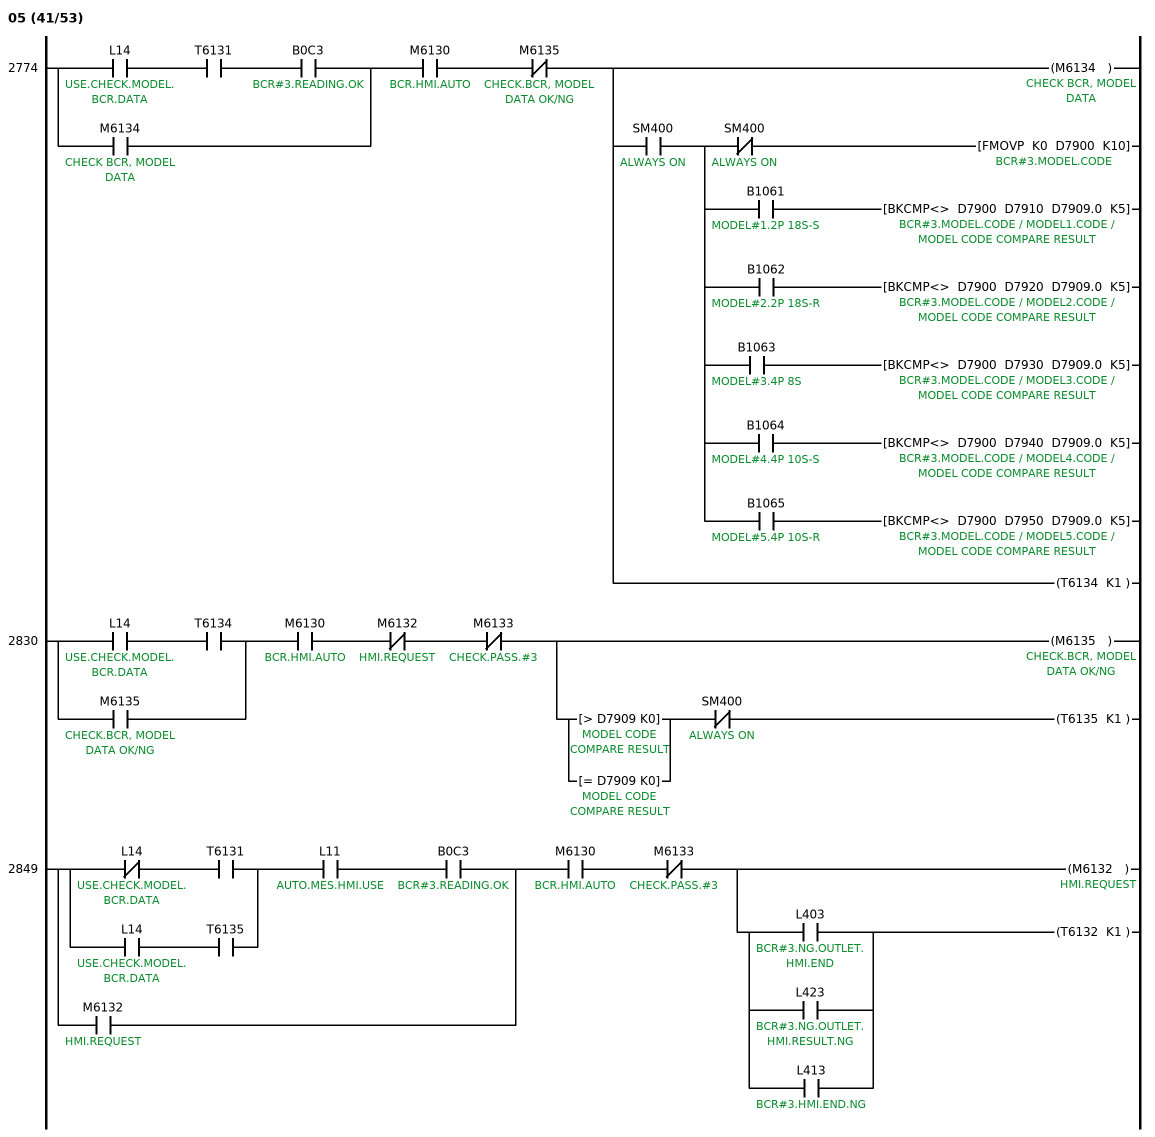
2774  LD      L14  ; USE.CHECK.MODEL.BCR.DATA
      AND     T6131
      AND     B0C3  ; BCR#3.READING.OK
      OR      M6134  ; CHECK BCR, MODEL DATA
      AND     M6130  ; BCR.HMI.AUTO
      ANI     M6135  ; CHECK.BCR, MODEL DATA OK/NG
      OUT     M6134  ; CHECK BCR, MODEL DATA
      MPS
      AND     SM400  ; ALWAYS ON
      MPS
      ANI     SM400  ; ALWAYS ON
      FMOVP   K0 D7900 K10  ; BCR#3.MODEL.CODE
      MRD
      AND     B1061  ; MODEL#1.2P 18S-S
      BKCMP<> D7900 D7910 D7909.0 K5  ; MODEL1.CODE / MODEL CODE COMPARE RESULT
      MRD
      AND     B1062  ; MODEL#2.2P 18S-R
      BKCMP<> D7900 D7920 D7909.0 K5  ; MODEL2.CODE
      MRD
      AND     B1063  ; MODEL#3.4P 8S
      BKCMP<> D7900 D7930 D7909.0 K5  ; MODEL3.CODE
      MRD
      AND     B1064  ; MODEL#4.4P 10S-S
      BKCMP<> D7900 D7940 D7909.0 K5  ; MODEL4.CODE
      MPP
      AND     B1065  ; MODEL#5.4P 10S-R
      BKCMP<> D7900 D7950 D7909.0 K5  ; MODEL5.CODE
      MPP
      OUT     T6134 K1
2830  LD      L14  ; USE.CHECK.MODEL.BCR.DATA
      AND     T6134
      OR      M6135  ; CHECK.BCR, MODEL DATA OK/NG
      AND     M6130  ; BCR.HMI.AUTO
      ANI     M6132  ; HMI.REQUEST
      ANI     M6133  ; CHECK.PASS.#3
      OUT     M6135  ; CHECK.BCR, MODEL DATA OK/NG
      LD>     D7909 K0  ; MODEL CODE COMPARE RESULT
      OR=     D7909 K0  ; MODEL CODE COMPARE RESULT
      ANB
      ANI     SM400  ; ALWAYS ON
      OUT     T6135 K1
2849  LDI     L14  ; USE.CHECK.MODEL.BCR.DATA
      AND     T6131
      LD      L14  ; USE.CHECK.MODEL.BCR.DATA
      AND     T6135
      ORB
      AND     L11  ; AUTO.MES.HMI.USE
      AND     B0C3  ; BCR#3.READING.OK
      OR      M6132  ; HMI.REQUEST
      AND     M6130  ; BCR.HMI.AUTO
      ANI     M6133  ; CHECK.PASS.#3
      OUT     M6132  ; HMI.REQUEST
      LD      L403  ; BCR#3.NG.OUTLET.HMI.END
      OR      L423  ; BCR#3.NG.OUTLET.HMI.RESULT.NG
      OR      L413  ; BCR#3.HMI.END.NG
      ANB
      OUT     T6132 K1
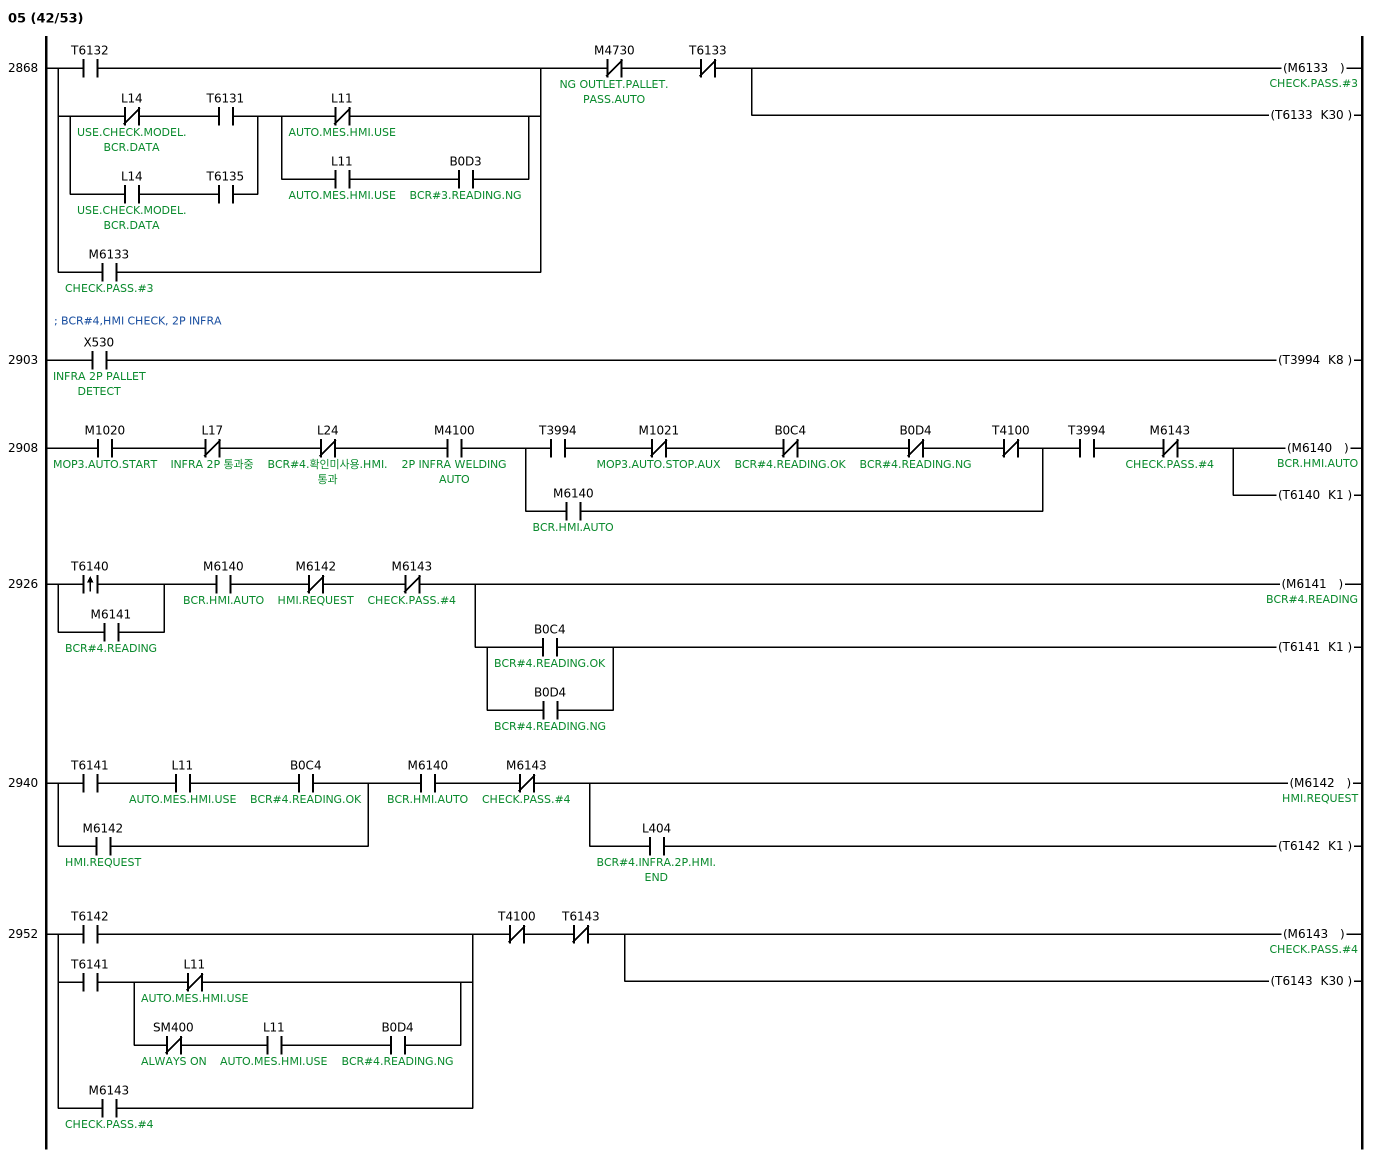
2868  LD      T6132
      LDI     L14  ; USE.CHECK.MODEL.BCR.DATA
      AND     T6131
      LD      L14  ; USE.CHECK.MODEL.BCR.DATA
      AND     T6135
      ORB
      LDI     L11  ; AUTO.MES.HMI.USE
      LD      L11  ; AUTO.MES.HMI.USE
      AND     B0D3  ; BCR#3.READING.NG
      ORB
      ANB
      ORB
      OR      M6133  ; CHECK.PASS.#3
      ANI     M4730  ; NG OUTLET.PALLET.PASS.AUTO
      ANI     T6133
      OUT     M6133  ; CHECK.PASS.#3
      OUT     T6133 K30
; BCR#4,HMI CHECK, 2P INFRA
2903  LD      X530  ; INFRA 2P PALLET DETECT
      OUT     T3994 K8
2908  LD      M1020  ; MOP3.AUTO.START
      ANI     L17  ; INFRA 2P 통과중
      ANI     L24  ; BCR#4.확인미사용.HMI.통과
      AND     M4100  ; 2P INFRA WELDING AUTO
      LD      T3994
      ANI     M1021  ; MOP3.AUTO.STOP.AUX
      ANI     B0C4  ; BCR#4.READING.OK
      ANI     B0D4  ; BCR#4.READING.NG
      ANI     T4100
      OR      M6140  ; BCR.HMI.AUTO
      ANB
      AND     T3994
      ANI     M6143  ; CHECK.PASS.#4
      OUT     M6140  ; BCR.HMI.AUTO
      OUT     T6140 K1
2926  LDP     T6140
      OR      M6141  ; BCR#4.READING
      AND     M6140  ; BCR.HMI.AUTO
      ANI     M6142  ; HMI.REQUEST
      ANI     M6143  ; CHECK.PASS.#4
      OUT     M6141  ; BCR#4.READING
      LD      B0C4  ; BCR#4.READING.OK
      OR      B0D4  ; BCR#4.READING.NG
      ANB
      OUT     T6141 K1
2940  LD      T6141
      AND     L11  ; AUTO.MES.HMI.USE
      AND     B0C4  ; BCR#4.READING.OK
      OR      M6142  ; HMI.REQUEST
      AND     M6140  ; BCR.HMI.AUTO
      ANI     M6143  ; CHECK.PASS.#4
      OUT     M6142  ; HMI.REQUEST
      AND     L404  ; BCR#4.INFRA.2P.HMI.END
      OUT     T6142 K1
2952  LD      T6142
      LD      T6141
      LDI     L11  ; AUTO.MES.HMI.USE
      LDI     SM400  ; ALWAYS ON
      AND     L11  ; AUTO.MES.HMI.USE
      AND     B0D4  ; BCR#4.READING.NG
      ORB
      ANB
      ORB
      OR      M6143  ; CHECK.PASS.#4
      ANI     T4100
      ANI     T6143
      OUT     M6143  ; CHECK.PASS.#4
      OUT     T6143 K30
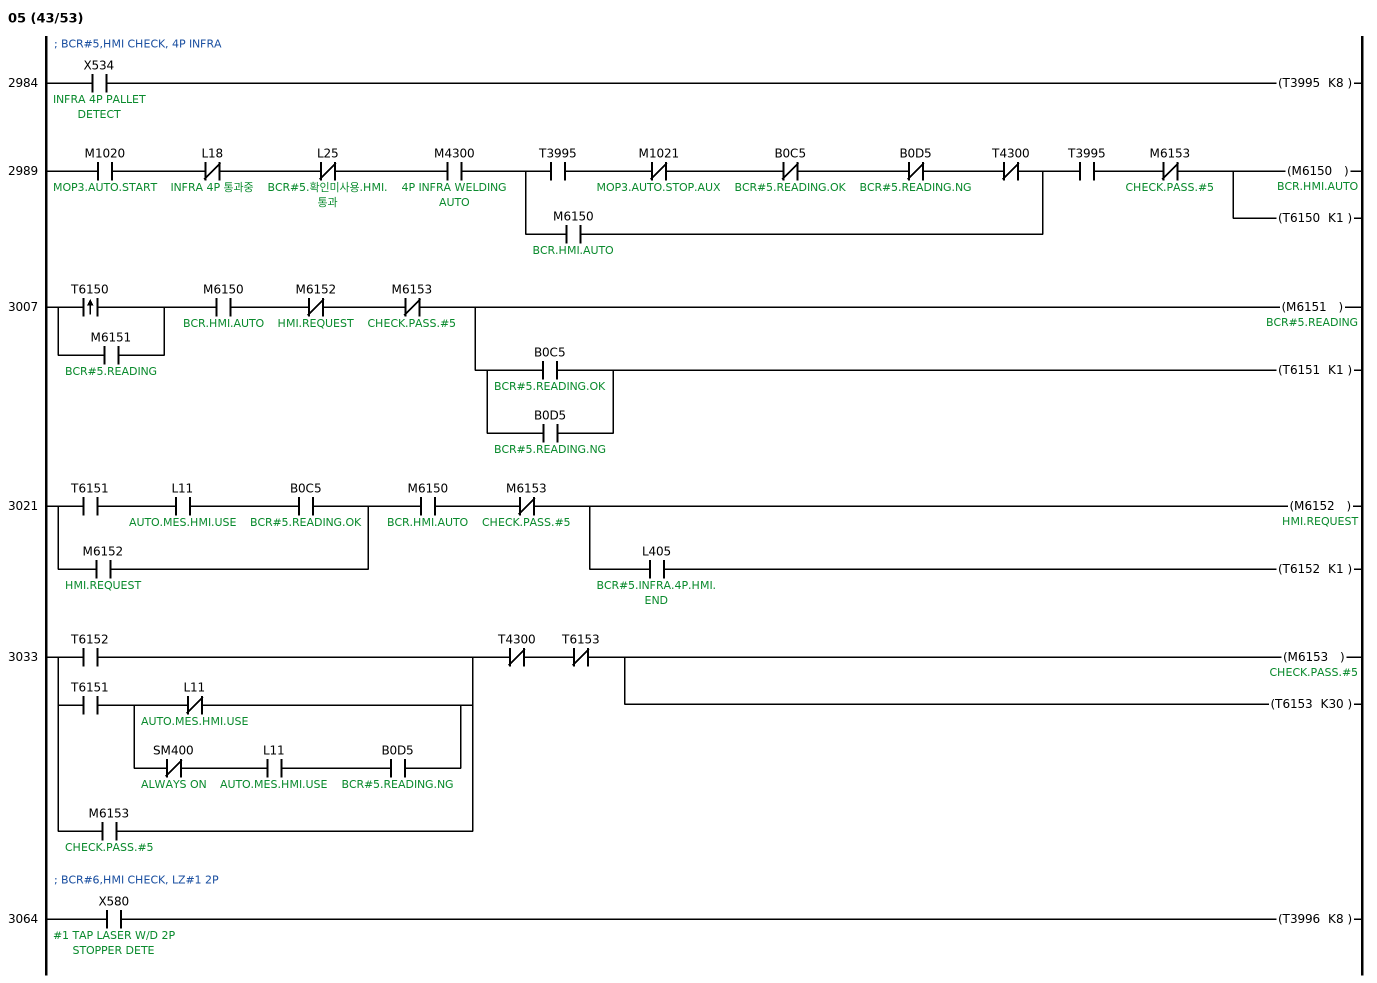
; BCR#5,HMI CHECK, 4P INFRA
2984  LD      X534  ; INFRA 4P PALLET DETECT
      OUT     T3995 K8
2989  LD      M1020  ; MOP3.AUTO.START
      ANI     L18  ; INFRA 4P 통과중
      ANI     L25  ; BCR#5.확인미사용.HMI.통과
      AND     M4300  ; 4P INFRA WELDING AUTO
      LD      T3995
      ANI     M1021  ; MOP3.AUTO.STOP.AUX
      ANI     B0C5  ; BCR#5.READING.OK
      ANI     B0D5  ; BCR#5.READING.NG
      ANI     T4300
      OR      M6150  ; BCR.HMI.AUTO
      ANB
      AND     T3995
      ANI     M6153  ; CHECK.PASS.#5
      OUT     M6150  ; BCR.HMI.AUTO
      OUT     T6150 K1
3007  LDP     T6150
      OR      M6151  ; BCR#5.READING
      AND     M6150  ; BCR.HMI.AUTO
      ANI     M6152  ; HMI.REQUEST
      ANI     M6153  ; CHECK.PASS.#5
      OUT     M6151  ; BCR#5.READING
      LD      B0C5  ; BCR#5.READING.OK
      OR      B0D5  ; BCR#5.READING.NG
      ANB
      OUT     T6151 K1
3021  LD      T6151
      AND     L11  ; AUTO.MES.HMI.USE
      AND     B0C5  ; BCR#5.READING.OK
      OR      M6152  ; HMI.REQUEST
      AND     M6150  ; BCR.HMI.AUTO
      ANI     M6153  ; CHECK.PASS.#5
      OUT     M6152  ; HMI.REQUEST
      AND     L405  ; BCR#5.INFRA.4P.HMI.END
      OUT     T6152 K1
3033  LD      T6152
      LD      T6151
      LDI     L11  ; AUTO.MES.HMI.USE
      LDI     SM400  ; ALWAYS ON
      AND     L11  ; AUTO.MES.HMI.USE
      AND     B0D5  ; BCR#5.READING.NG
      ORB
      ANB
      ORB
      OR      M6153  ; CHECK.PASS.#5
      ANI     T4300
      ANI     T6153
      OUT     M6153  ; CHECK.PASS.#5
      OUT     T6153 K30
; BCR#6,HMI CHECK, LZ#1 2P
3064  LD      X580  ; #1 TAP LASER W/D 2P STOPPER DETE
      OUT     T3996 K8
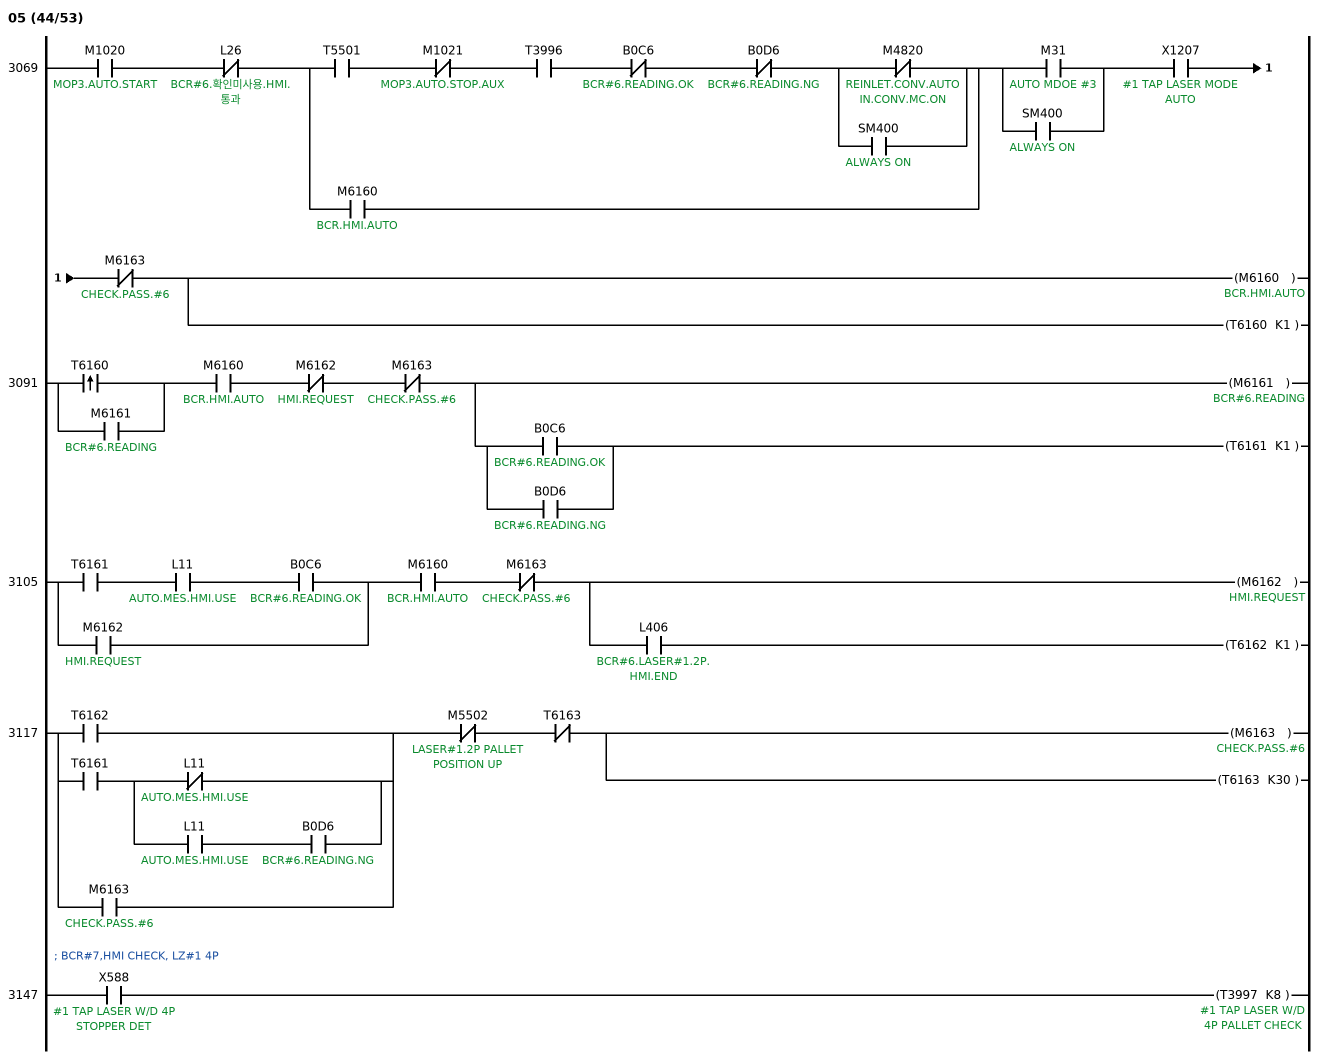
3069  LD      M1020  ; MOP3.AUTO.START
      ANI     L26  ; BCR#6.확인미사용.HMI.통과
      LD      T5501
      ANI     M1021  ; MOP3.AUTO.STOP.AUX
      AND     T3996
      ANI     B0C6  ; BCR#6.READING.OK
      ANI     B0D6  ; BCR#6.READING.NG
      LDI     M4820  ; REINLET.CONV.AUTO IN.CONV.MC.ON
      OR      SM400  ; ALWAYS ON
      ANB
      OR      M6160  ; BCR.HMI.AUTO
      ANB
      LD      M31  ; AUTO MDOE #3
      OR      SM400  ; ALWAYS ON
      ANB
      AND     X1207  ; #1 TAP LASER MODE AUTO
      ANI     M6163  ; CHECK.PASS.#6
      OUT     M6160  ; BCR.HMI.AUTO
      OUT     T6160 K1
3091  LDP     T6160
      OR      M6161  ; BCR#6.READING
      AND     M6160  ; BCR.HMI.AUTO
      ANI     M6162  ; HMI.REQUEST
      ANI     M6163  ; CHECK.PASS.#6
      OUT     M6161  ; BCR#6.READING
      LD      B0C6  ; BCR#6.READING.OK
      OR      B0D6  ; BCR#6.READING.NG
      ANB
      OUT     T6161 K1
3105  LD      T6161
      AND     L11  ; AUTO.MES.HMI.USE
      AND     B0C6  ; BCR#6.READING.OK
      OR      M6162  ; HMI.REQUEST
      AND     M6160  ; BCR.HMI.AUTO
      ANI     M6163  ; CHECK.PASS.#6
      OUT     M6162  ; HMI.REQUEST
      AND     L406  ; BCR#6.LASER#1.2P.HMI.END
      OUT     T6162 K1
3117  LD      T6162
      LD      T6161
      LDI     L11  ; AUTO.MES.HMI.USE
      LD      L11  ; AUTO.MES.HMI.USE
      AND     B0D6  ; BCR#6.READING.NG
      ORB
      ANB
      ORB
      OR      M6163  ; CHECK.PASS.#6
      ANI     M5502  ; LASER#1.2P PALLET POSITION UP
      ANI     T6163
      OUT     M6163  ; CHECK.PASS.#6
      OUT     T6163 K30
; BCR#7,HMI CHECK, LZ#1 4P
3147  LD      X588  ; #1 TAP LASER W/D 4P STOPPER DET
      OUT     T3997 K8  ; #1 TAP LASER W/D 4P PALLET CHECK
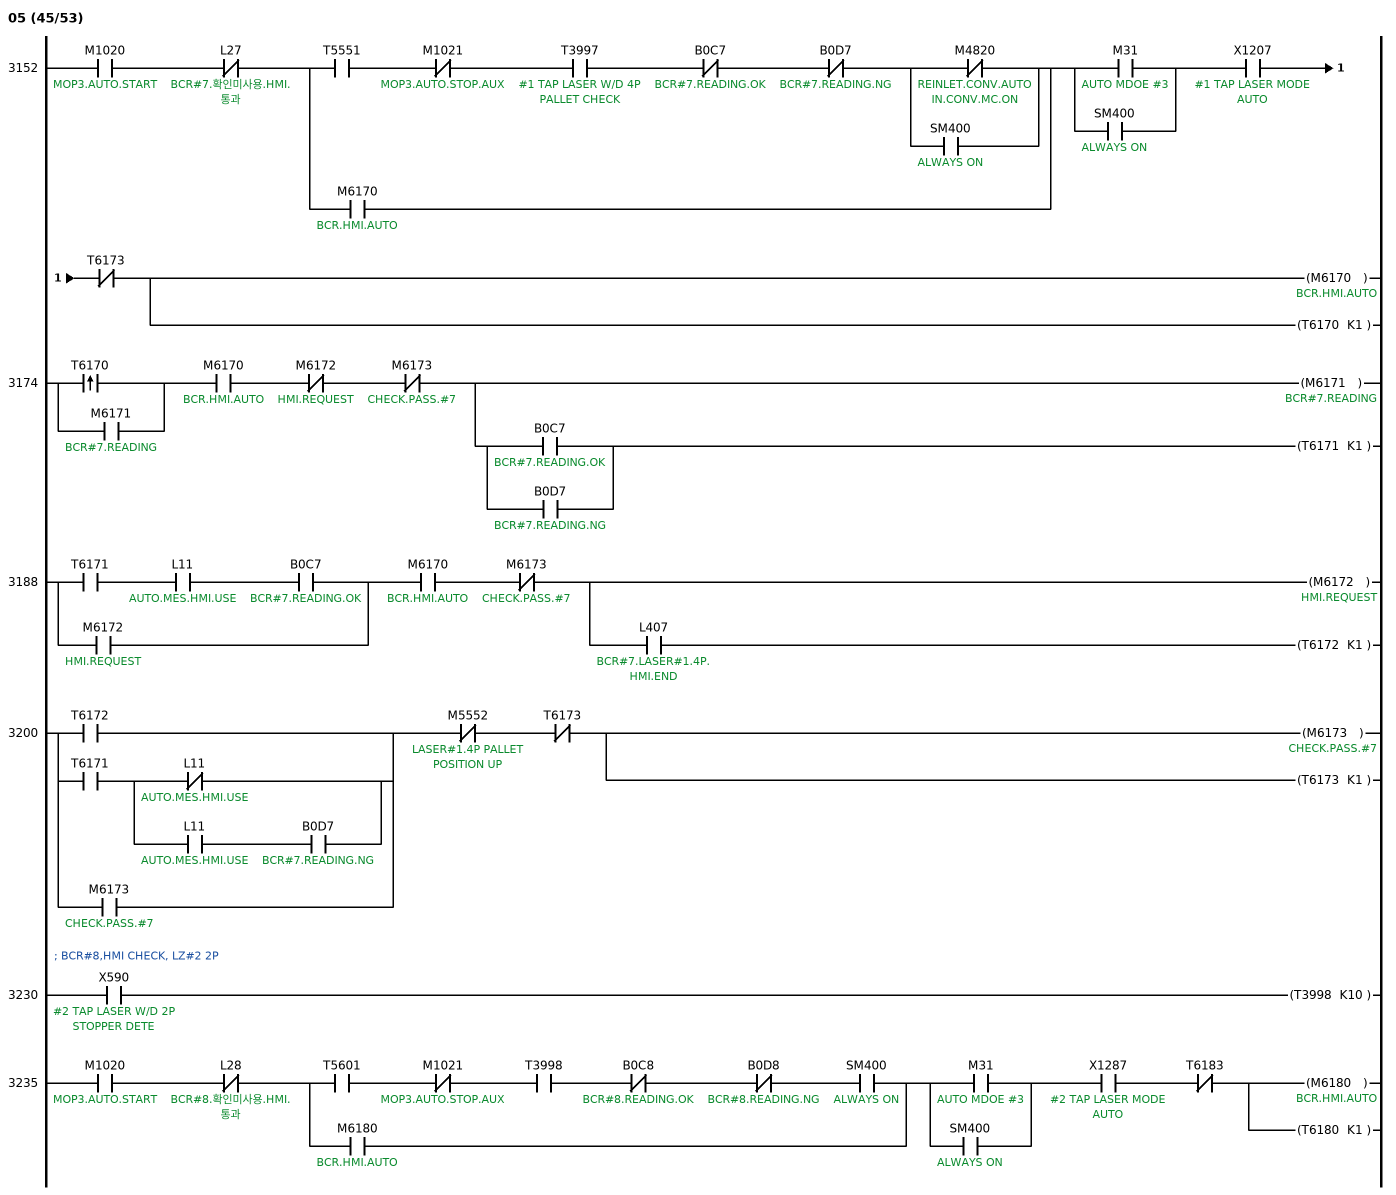
3152  LD      M1020  ; MOP3.AUTO.START
      ANI     L27  ; BCR#7.확인미사용.HMI.통과
      LD      T5551
      ANI     M1021  ; MOP3.AUTO.STOP.AUX
      AND     T3997  ; #1 TAP LASER W/D 4P PALLET CHECK
      ANI     B0C7  ; BCR#7.READING.OK
      ANI     B0D7  ; BCR#7.READING.NG
      LDI     M4820  ; REINLET.CONV.AUTO IN.CONV.MC.ON
      OR      SM400  ; ALWAYS ON
      ANB
      OR      M6170  ; BCR.HMI.AUTO
      ANB
      LD      M31  ; AUTO MDOE #3
      OR      SM400  ; ALWAYS ON
      ANB
      AND     X1207  ; #1 TAP LASER MODE AUTO
      ANI     T6173
      OUT     M6170  ; BCR.HMI.AUTO
      OUT     T6170 K1
3174  LDP     T6170
      OR      M6171  ; BCR#7.READING
      AND     M6170  ; BCR.HMI.AUTO
      ANI     M6172  ; HMI.REQUEST
      ANI     M6173  ; CHECK.PASS.#7
      OUT     M6171  ; BCR#7.READING
      LD      B0C7  ; BCR#7.READING.OK
      OR      B0D7  ; BCR#7.READING.NG
      ANB
      OUT     T6171 K1
3188  LD      T6171
      AND     L11  ; AUTO.MES.HMI.USE
      AND     B0C7  ; BCR#7.READING.OK
      OR      M6172  ; HMI.REQUEST
      AND     M6170  ; BCR.HMI.AUTO
      ANI     M6173  ; CHECK.PASS.#7
      OUT     M6172  ; HMI.REQUEST
      AND     L407  ; BCR#7.LASER#1.4P.HMI.END
      OUT     T6172 K1
3200  LD      T6172
      LD      T6171
      LDI     L11  ; AUTO.MES.HMI.USE
      LD      L11  ; AUTO.MES.HMI.USE
      AND     B0D7  ; BCR#7.READING.NG
      ORB
      ANB
      ORB
      OR      M6173  ; CHECK.PASS.#7
      ANI     M5552  ; LASER#1.4P PALLET POSITION UP
      ANI     T6173
      OUT     M6173  ; CHECK.PASS.#7
      OUT     T6173 K1
; BCR#8,HMI CHECK, LZ#2 2P
3230  LD      X590  ; #2 TAP LASER W/D 2P STOPPER DETE
      OUT     T3998 K10
3235  LD      M1020  ; MOP3.AUTO.START
      ANI     L28  ; BCR#8.확인미사용.HMI.통과
      LD      T5601
      ANI     M1021  ; MOP3.AUTO.STOP.AUX
      AND     T3998
      ANI     B0C8  ; BCR#8.READING.OK
      ANI     B0D8  ; BCR#8.READING.NG
      AND     SM400  ; ALWAYS ON
      OR      M6180  ; BCR.HMI.AUTO
      ANB
      LD      M31  ; AUTO MDOE #3
      OR      SM400  ; ALWAYS ON
      ANB
      AND     X1287  ; #2 TAP LASER MODE AUTO
      ANI     T6183
      OUT     M6180  ; BCR.HMI.AUTO
      OUT     T6180 K1
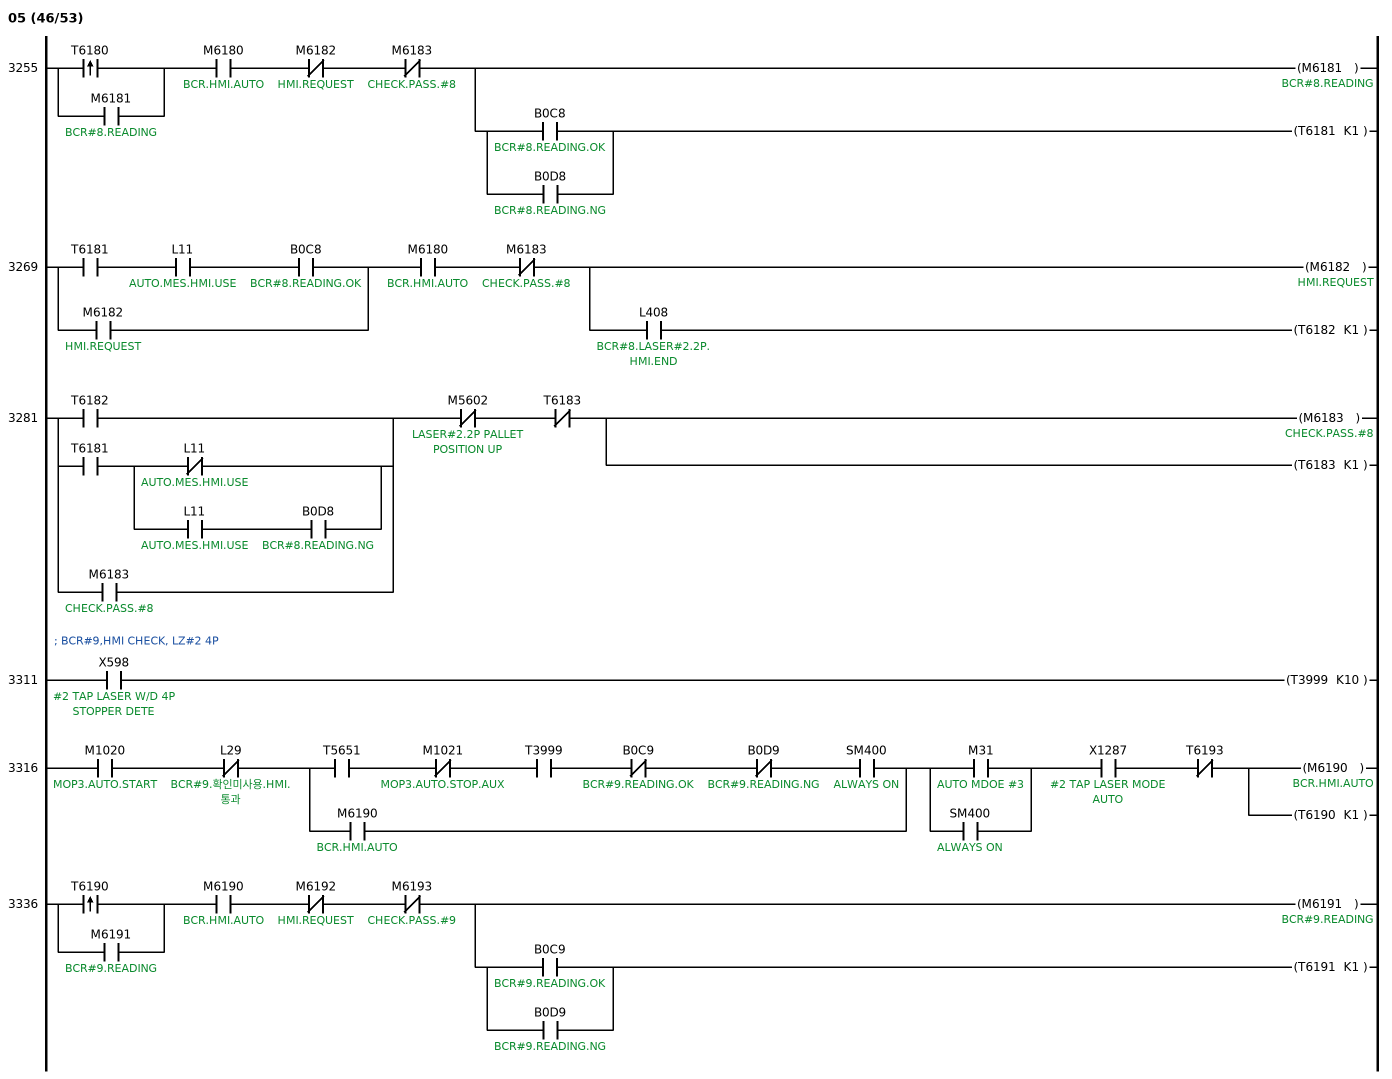
3255  LDP     T6180
      OR      M6181  ; BCR#8.READING
      AND     M6180  ; BCR.HMI.AUTO
      ANI     M6182  ; HMI.REQUEST
      ANI     M6183  ; CHECK.PASS.#8
      OUT     M6181  ; BCR#8.READING
      LD      B0C8  ; BCR#8.READING.OK
      OR      B0D8  ; BCR#8.READING.NG
      ANB
      OUT     T6181 K1
3269  LD      T6181
      AND     L11  ; AUTO.MES.HMI.USE
      AND     B0C8  ; BCR#8.READING.OK
      OR      M6182  ; HMI.REQUEST
      AND     M6180  ; BCR.HMI.AUTO
      ANI     M6183  ; CHECK.PASS.#8
      OUT     M6182  ; HMI.REQUEST
      AND     L408  ; BCR#8.LASER#2.2P.HMI.END
      OUT     T6182 K1
3281  LD      T6182
      LD      T6181
      LDI     L11  ; AUTO.MES.HMI.USE
      LD      L11  ; AUTO.MES.HMI.USE
      AND     B0D8  ; BCR#8.READING.NG
      ORB
      ANB
      ORB
      OR      M6183  ; CHECK.PASS.#8
      ANI     M5602  ; LASER#2.2P PALLET POSITION UP
      ANI     T6183
      OUT     M6183  ; CHECK.PASS.#8
      OUT     T6183 K1
; BCR#9,HMI CHECK, LZ#2 4P
3311  LD      X598  ; #2 TAP LASER W/D 4P STOPPER DETE
      OUT     T3999 K10
3316  LD      M1020  ; MOP3.AUTO.START
      ANI     L29  ; BCR#9.확인미사용.HMI.통과
      LD      T5651
      ANI     M1021  ; MOP3.AUTO.STOP.AUX
      AND     T3999
      ANI     B0C9  ; BCR#9.READING.OK
      ANI     B0D9  ; BCR#9.READING.NG
      AND     SM400  ; ALWAYS ON
      OR      M6190  ; BCR.HMI.AUTO
      ANB
      LD      M31  ; AUTO MDOE #3
      OR      SM400  ; ALWAYS ON
      ANB
      AND     X1287  ; #2 TAP LASER MODE AUTO
      ANI     T6193
      OUT     M6190  ; BCR.HMI.AUTO
      OUT     T6190 K1
3336  LDP     T6190
      OR      M6191  ; BCR#9.READING
      AND     M6190  ; BCR.HMI.AUTO
      ANI     M6192  ; HMI.REQUEST
      ANI     M6193  ; CHECK.PASS.#9
      OUT     M6191  ; BCR#9.READING
      LD      B0C9  ; BCR#9.READING.OK
      OR      B0D9  ; BCR#9.READING.NG
      ANB
      OUT     T6191 K1
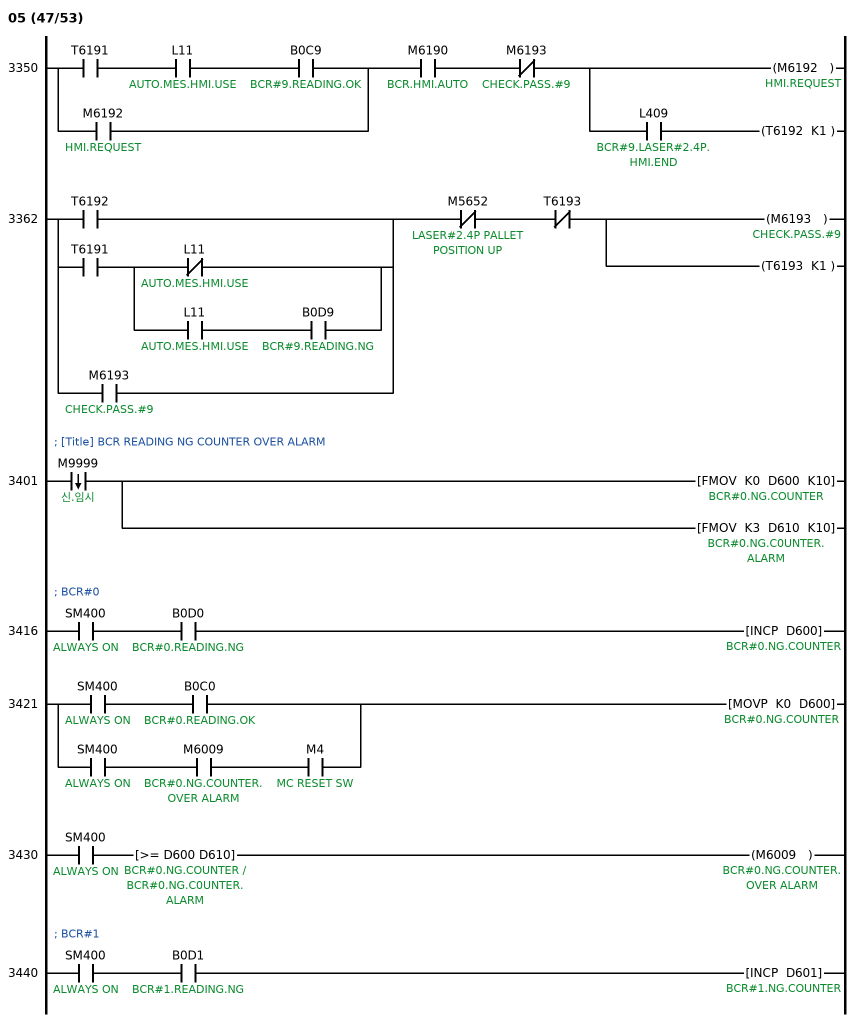
3350  LD      T6191
      AND     L11  ; AUTO.MES.HMI.USE
      AND     B0C9  ; BCR#9.READING.OK
      OR      M6192  ; HMI.REQUEST
      AND     M6190  ; BCR.HMI.AUTO
      ANI     M6193  ; CHECK.PASS.#9
      OUT     M6192  ; HMI.REQUEST
      AND     L409  ; BCR#9.LASER#2.4P.HMI.END
      OUT     T6192 K1
3362  LD      T6192
      LD      T6191
      LDI     L11  ; AUTO.MES.HMI.USE
      LD      L11  ; AUTO.MES.HMI.USE
      AND     B0D9  ; BCR#9.READING.NG
      ORB
      ANB
      ORB
      OR      M6193  ; CHECK.PASS.#9
      ANI     M5652  ; LASER#2.4P PALLET POSITION UP
      ANI     T6193
      OUT     M6193  ; CHECK.PASS.#9
      OUT     T6193 K1
; [Title] BCR READING NG COUNTER OVER ALARM
3401  LDF     M9999  ; 신.임시
      FMOV    K0 D600 K10  ; BCR#0.NG.COUNTER
      FMOV    K3 D610 K10  ; BCR#0.NG.C0UNTER.ALARM
; BCR#0
3416  LD      SM400  ; ALWAYS ON
      AND     B0D0  ; BCR#0.READING.NG
      INCP    D600
3421  LD      SM400  ; ALWAYS ON
      AND     B0C0  ; BCR#0.READING.OK
      LD      SM400  ; ALWAYS ON
      AND     M6009  ; BCR#0.NG.COUNTER.OVER ALARM
      AND     M4  ; MC RESET SW
      ORB
      MOVP    K0 D600
3430  LD      SM400  ; ALWAYS ON
      AND>=   D600 D610  ; BCR#0.NG.COUNTER / BCR#0.NG.C0UNTER.ALARM
      OUT     M6009  ; BCR#0.NG.COUNTER.OVER ALARM
; BCR#1
3440  LD      SM400  ; ALWAYS ON
      AND     B0D1  ; BCR#1.READING.NG
      INCP    D601  ; BCR#1.NG.COUNTER
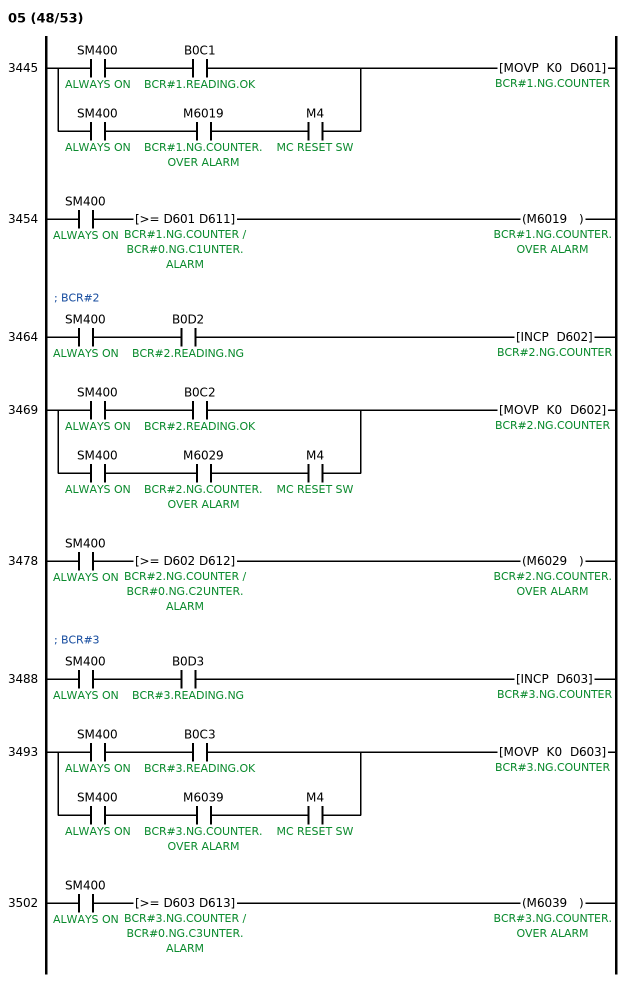
3445  LD      SM400  ; ALWAYS ON
      AND     B0C1  ; BCR#1.READING.OK
      LD      SM400  ; ALWAYS ON
      AND     M6019  ; BCR#1.NG.COUNTER.OVER ALARM
      AND     M4  ; MC RESET SW
      ORB
      MOVP    K0 D601
3454  LD      SM400  ; ALWAYS ON
      AND>=   D601 D611  ; BCR#1.NG.COUNTER / BCR#0.NG.C1UNTER.ALARM
      OUT     M6019  ; BCR#1.NG.COUNTER.OVER ALARM
; BCR#2
3464  LD      SM400  ; ALWAYS ON
      AND     B0D2  ; BCR#2.READING.NG
      INCP    D602  ; BCR#2.NG.COUNTER
3469  LD      SM400  ; ALWAYS ON
      AND     B0C2  ; BCR#2.READING.OK
      LD      SM400  ; ALWAYS ON
      AND     M6029  ; BCR#2.NG.COUNTER.OVER ALARM
      AND     M4  ; MC RESET SW
      ORB
      MOVP    K0 D602
3478  LD      SM400  ; ALWAYS ON
      AND>=   D602 D612  ; BCR#2.NG.COUNTER / BCR#0.NG.C2UNTER.ALARM
      OUT     M6029  ; BCR#2.NG.COUNTER.OVER ALARM
; BCR#3
3488  LD      SM400  ; ALWAYS ON
      AND     B0D3  ; BCR#3.READING.NG
      INCP    D603  ; BCR#3.NG.COUNTER
3493  LD      SM400  ; ALWAYS ON
      AND     B0C3  ; BCR#3.READING.OK
      LD      SM400  ; ALWAYS ON
      AND     M6039  ; BCR#3.NG.COUNTER.OVER ALARM
      AND     M4  ; MC RESET SW
      ORB
      MOVP    K0 D603
3502  LD      SM400  ; ALWAYS ON
      AND>=   D603 D613  ; BCR#3.NG.COUNTER / BCR#0.NG.C3UNTER.ALARM
      OUT     M6039  ; BCR#3.NG.COUNTER.OVER ALARM
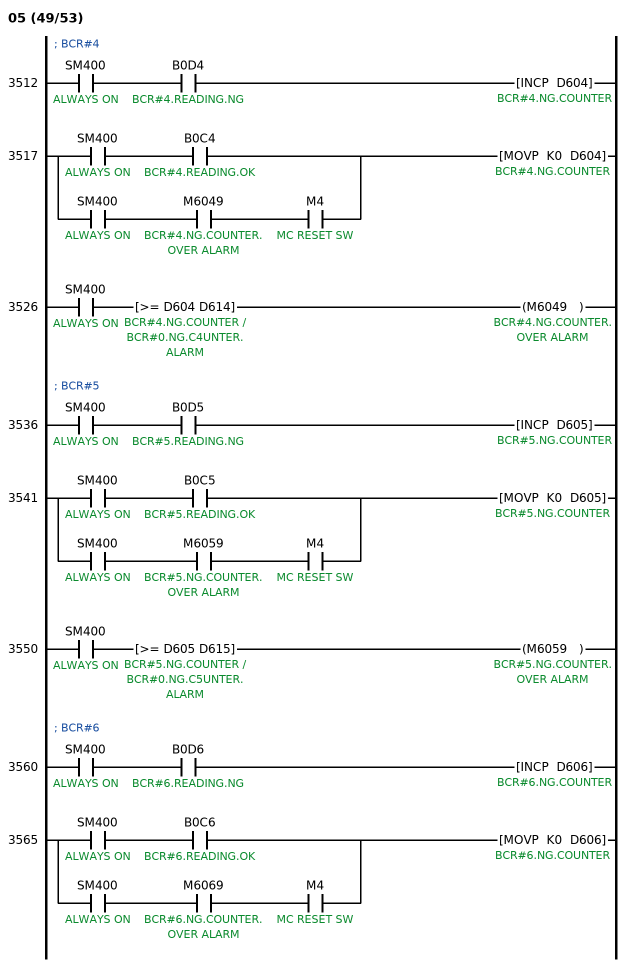
; BCR#4
3512  LD      SM400  ; ALWAYS ON
      AND     B0D4  ; BCR#4.READING.NG
      INCP    D604  ; BCR#4.NG.COUNTER
3517  LD      SM400  ; ALWAYS ON
      AND     B0C4  ; BCR#4.READING.OK
      LD      SM400  ; ALWAYS ON
      AND     M6049  ; BCR#4.NG.COUNTER.OVER ALARM
      AND     M4  ; MC RESET SW
      ORB
      MOVP    K0 D604
3526  LD      SM400  ; ALWAYS ON
      AND>=   D604 D614  ; BCR#4.NG.COUNTER / BCR#0.NG.C4UNTER.ALARM
      OUT     M6049  ; BCR#4.NG.COUNTER.OVER ALARM
; BCR#5
3536  LD      SM400  ; ALWAYS ON
      AND     B0D5  ; BCR#5.READING.NG
      INCP    D605  ; BCR#5.NG.COUNTER
3541  LD      SM400  ; ALWAYS ON
      AND     B0C5  ; BCR#5.READING.OK
      LD      SM400  ; ALWAYS ON
      AND     M6059  ; BCR#5.NG.COUNTER.OVER ALARM
      AND     M4  ; MC RESET SW
      ORB
      MOVP    K0 D605
3550  LD      SM400  ; ALWAYS ON
      AND>=   D605 D615  ; BCR#5.NG.COUNTER / BCR#0.NG.C5UNTER.ALARM
      OUT     M6059  ; BCR#5.NG.COUNTER.OVER ALARM
; BCR#6
3560  LD      SM400  ; ALWAYS ON
      AND     B0D6  ; BCR#6.READING.NG
      INCP    D606  ; BCR#6.NG.COUNTER
3565  LD      SM400  ; ALWAYS ON
      AND     B0C6  ; BCR#6.READING.OK
      LD      SM400  ; ALWAYS ON
      AND     M6069  ; BCR#6.NG.COUNTER.OVER ALARM
      AND     M4  ; MC RESET SW
      ORB
      MOVP    K0 D606
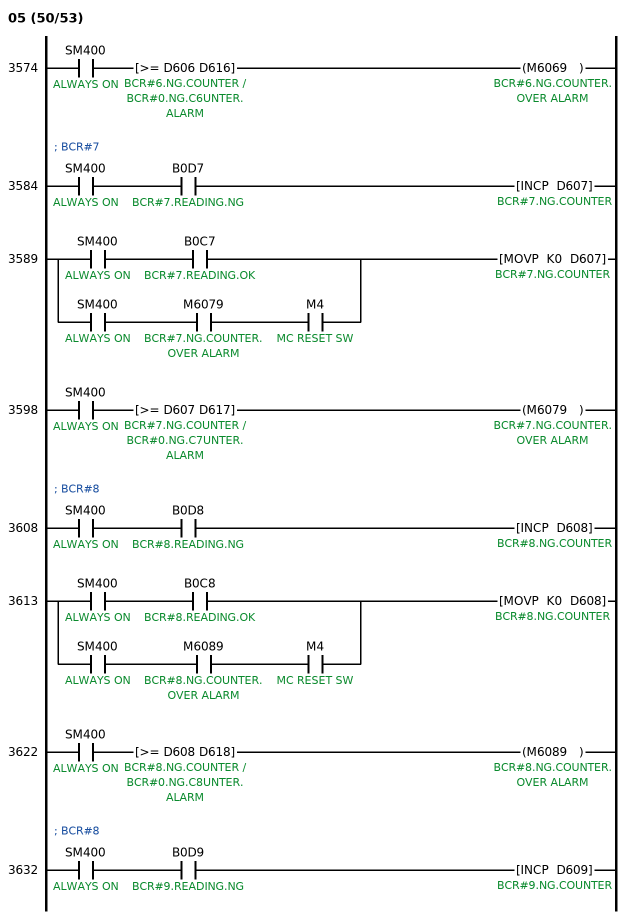
3574  LD      SM400  ; ALWAYS ON
      AND>=   D606 D616  ; BCR#6.NG.COUNTER / BCR#0.NG.C6UNTER.ALARM
      OUT     M6069  ; BCR#6.NG.COUNTER.OVER ALARM
; BCR#7
3584  LD      SM400  ; ALWAYS ON
      AND     B0D7  ; BCR#7.READING.NG
      INCP    D607  ; BCR#7.NG.COUNTER
3589  LD      SM400  ; ALWAYS ON
      AND     B0C7  ; BCR#7.READING.OK
      LD      SM400  ; ALWAYS ON
      AND     M6079  ; BCR#7.NG.COUNTER.OVER ALARM
      AND     M4  ; MC RESET SW
      ORB
      MOVP    K0 D607
3598  LD      SM400  ; ALWAYS ON
      AND>=   D607 D617  ; BCR#7.NG.COUNTER / BCR#0.NG.C7UNTER.ALARM
      OUT     M6079  ; BCR#7.NG.COUNTER.OVER ALARM
; BCR#8
3608  LD      SM400  ; ALWAYS ON
      AND     B0D8  ; BCR#8.READING.NG
      INCP    D608  ; BCR#8.NG.COUNTER
3613  LD      SM400  ; ALWAYS ON
      AND     B0C8  ; BCR#8.READING.OK
      LD      SM400  ; ALWAYS ON
      AND     M6089  ; BCR#8.NG.COUNTER.OVER ALARM
      AND     M4  ; MC RESET SW
      ORB
      MOVP    K0 D608
3622  LD      SM400  ; ALWAYS ON
      AND>=   D608 D618  ; BCR#8.NG.COUNTER / BCR#0.NG.C8UNTER.ALARM
      OUT     M6089  ; BCR#8.NG.COUNTER.OVER ALARM
; BCR#8
3632  LD      SM400  ; ALWAYS ON
      AND     B0D9  ; BCR#9.READING.NG
      INCP    D609  ; BCR#9.NG.COUNTER
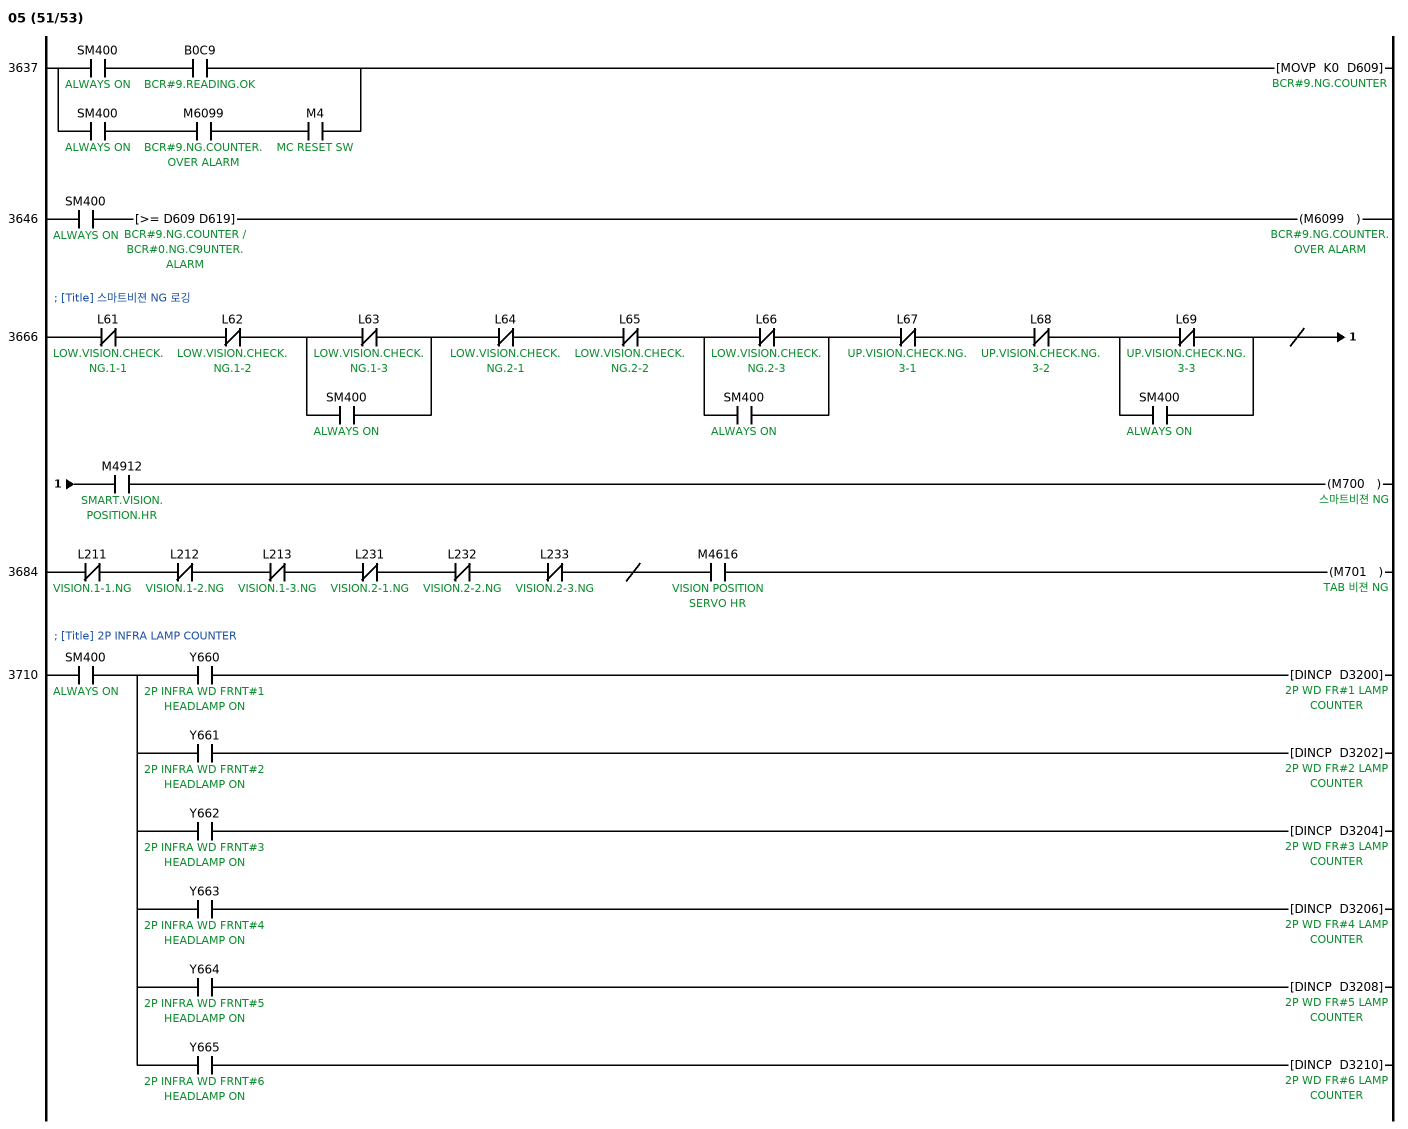
3637  LD      SM400  ; ALWAYS ON
      AND     B0C9  ; BCR#9.READING.OK
      LD      SM400  ; ALWAYS ON
      AND     M6099  ; BCR#9.NG.COUNTER.OVER ALARM
      AND     M4  ; MC RESET SW
      ORB
      MOVP    K0 D609
3646  LD      SM400  ; ALWAYS ON
      AND>=   D609 D619  ; BCR#9.NG.COUNTER / BCR#0.NG.C9UNTER.ALARM
      OUT     M6099  ; BCR#9.NG.COUNTER.OVER ALARM
; [Title] 스마트비젼 NG 로깅
3666  LDI     L61  ; LOW.VISION.CHECK.NG.1-1
      ANI     L62  ; LOW.VISION.CHECK.NG.1-2
      LDI     L63  ; LOW.VISION.CHECK.NG.1-3
      OR      SM400  ; ALWAYS ON
      ANB
      ANI     L64  ; LOW.VISION.CHECK.NG.2-1
      ANI     L65  ; LOW.VISION.CHECK.NG.2-2
      LDI     L66  ; LOW.VISION.CHECK.NG.2-3
      OR      SM400  ; ALWAYS ON
      ANB
      ANI     L67  ; UP.VISION.CHECK.NG.3-1
      ANI     L68  ; UP.VISION.CHECK.NG.3-2
      LDI     L69  ; UP.VISION.CHECK.NG.3-3
      OR      SM400  ; ALWAYS ON
      ANB
      INV
      AND     M4912  ; SMART.VISION.POSITION.HR
      OUT     M700  ; 스마트비젼 NG
3684  LDI     L211  ; VISION.1-1.NG
      ANI     L212  ; VISION.1-2.NG
      ANI     L213  ; VISION.1-3.NG
      ANI     L231  ; VISION.2-1.NG
      ANI     L232  ; VISION.2-2.NG
      ANI     L233  ; VISION.2-3.NG
      INV
      AND     M4616  ; VISION POSITION SERVO HR
      OUT     M701  ; TAB 비젼 NG
; [Title] 2P INFRA LAMP COUNTER
3710  LD      SM400  ; ALWAYS ON
      MPS
      AND     Y660  ; 2P INFRA WD FRNT#1 HEADLAMP ON
      DINCP   D3200  ; 2P WD FR#1 LAMP COUNTER
      MRD
      AND     Y661  ; 2P INFRA WD FRNT#2 HEADLAMP ON
      DINCP   D3202  ; 2P WD FR#2 LAMP COUNTER
      MRD
      AND     Y662  ; 2P INFRA WD FRNT#3 HEADLAMP ON
      DINCP   D3204  ; 2P WD FR#3 LAMP COUNTER
      MRD
      AND     Y663  ; 2P INFRA WD FRNT#4 HEADLAMP ON
      DINCP   D3206  ; 2P WD FR#4 LAMP COUNTER
      MRD
      AND     Y664  ; 2P INFRA WD FRNT#5 HEADLAMP ON
      DINCP   D3208  ; 2P WD FR#5 LAMP COUNTER
      MPP
      AND     Y665  ; 2P INFRA WD FRNT#6 HEADLAMP ON
      DINCP   D3210  ; 2P WD FR#6 LAMP COUNTER
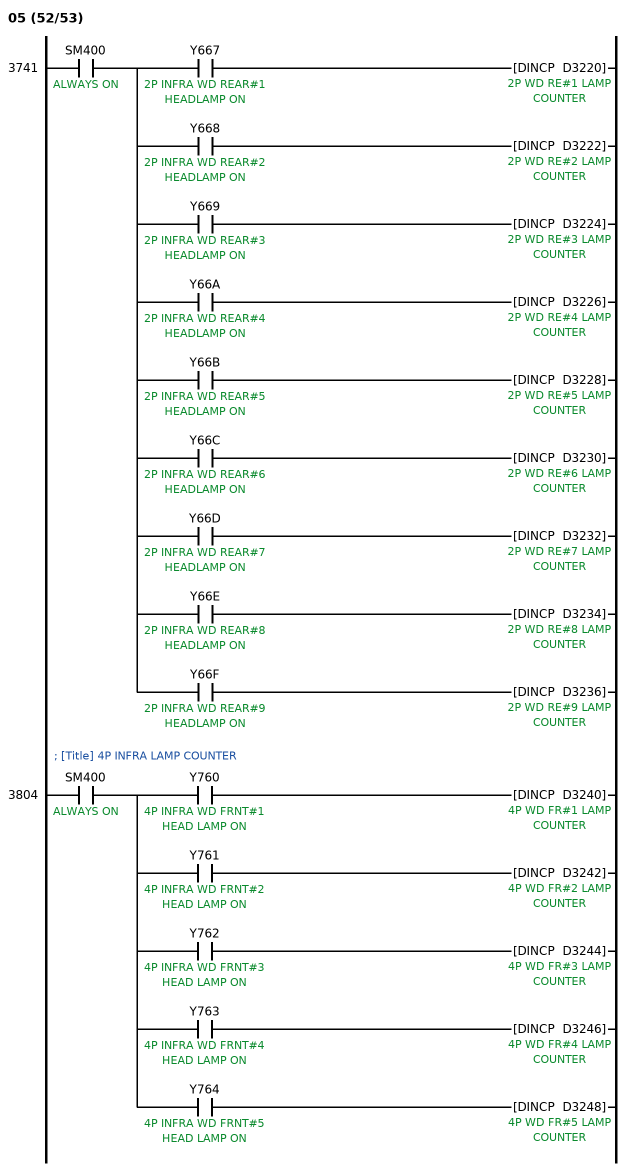
3741  LD      SM400  ; ALWAYS ON
      MPS
      AND     Y667  ; 2P INFRA WD REAR#1 HEADLAMP ON
      DINCP   D3220  ; 2P WD RE#1 LAMP COUNTER
      MRD
      AND     Y668  ; 2P INFRA WD REAR#2 HEADLAMP ON
      DINCP   D3222  ; 2P WD RE#2 LAMP COUNTER
      MRD
      AND     Y669  ; 2P INFRA WD REAR#3 HEADLAMP ON
      DINCP   D3224  ; 2P WD RE#3 LAMP COUNTER
      MRD
      AND     Y66A  ; 2P INFRA WD REAR#4 HEADLAMP ON
      DINCP   D3226  ; 2P WD RE#4 LAMP COUNTER
      MRD
      AND     Y66B  ; 2P INFRA WD REAR#5 HEADLAMP ON
      DINCP   D3228  ; 2P WD RE#5 LAMP COUNTER
      MRD
      AND     Y66C  ; 2P INFRA WD REAR#6 HEADLAMP ON
      DINCP   D3230  ; 2P WD RE#6 LAMP COUNTER
      MRD
      AND     Y66D  ; 2P INFRA WD REAR#7 HEADLAMP ON
      DINCP   D3232  ; 2P WD RE#7 LAMP COUNTER
      MRD
      AND     Y66E  ; 2P INFRA WD REAR#8 HEADLAMP ON
      DINCP   D3234  ; 2P WD RE#8 LAMP COUNTER
      MPP
      AND     Y66F  ; 2P INFRA WD REAR#9 HEADLAMP ON
      DINCP   D3236  ; 2P WD RE#9 LAMP COUNTER
; [Title] 4P INFRA LAMP COUNTER
3804  LD      SM400  ; ALWAYS ON
      MPS
      AND     Y760  ; 4P INFRA WD FRNT#1 HEAD LAMP ON
      DINCP   D3240  ; 4P WD FR#1 LAMP COUNTER
      MRD
      AND     Y761  ; 4P INFRA WD FRNT#2 HEAD LAMP ON
      DINCP   D3242  ; 4P WD FR#2 LAMP COUNTER
      MRD
      AND     Y762  ; 4P INFRA WD FRNT#3 HEAD LAMP ON
      DINCP   D3244  ; 4P WD FR#3 LAMP COUNTER
      MRD
      AND     Y763  ; 4P INFRA WD FRNT#4 HEAD LAMP ON
      DINCP   D3246  ; 4P WD FR#4 LAMP COUNTER
      MPP
      AND     Y764  ; 4P INFRA WD FRNT#5 HEAD LAMP ON
      DINCP   D3248  ; 4P WD FR#5 LAMP COUNTER
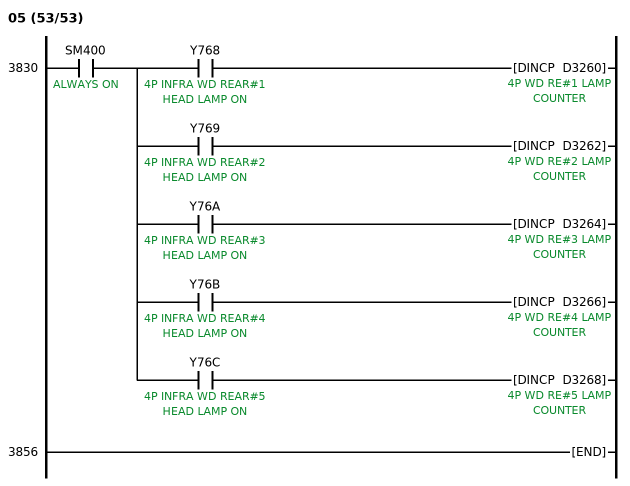
3830  LD      SM400  ; ALWAYS ON
      MPS
      AND     Y768  ; 4P INFRA WD REAR#1 HEAD LAMP ON
      DINCP   D3260  ; 4P WD RE#1 LAMP COUNTER
      MRD
      AND     Y769  ; 4P INFRA WD REAR#2 HEAD LAMP ON
      DINCP   D3262  ; 4P WD RE#2 LAMP COUNTER
      MRD
      AND     Y76A  ; 4P INFRA WD REAR#3 HEAD LAMP ON
      DINCP   D3264  ; 4P WD RE#3 LAMP COUNTER
      MRD
      AND     Y76B  ; 4P INFRA WD REAR#4 HEAD LAMP ON
      DINCP   D3266  ; 4P WD RE#4 LAMP COUNTER
      MPP
      AND     Y76C  ; 4P INFRA WD REAR#5 HEAD LAMP ON
      DINCP   D3268  ; 4P WD RE#5 LAMP COUNTER
3856  END
END_PROGRAM

PROGRAM 11  // SERVO DATA (1)
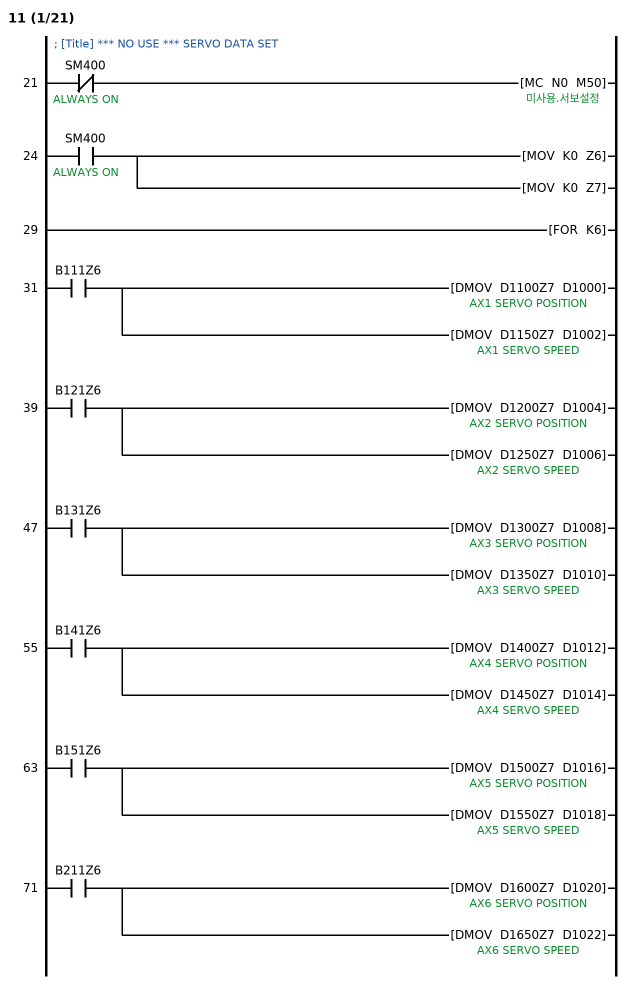
; [Title] *** NO USE *** SERVO DATA SET
21    LDI     SM400  ; ALWAYS ON
      MC      N0 M50  ; 미사용.서보설정
24    LD      SM400  ; ALWAYS ON
      MOV     K0 Z6
      MOV     K0 Z7
29    FOR     K6
31    LD      B111Z6
      DMOV    D1100Z7 D1000  ; AX1 SERVO POSITION
      DMOV    D1150Z7 D1002  ; AX1 SERVO SPEED
39    LD      B121Z6
      DMOV    D1200Z7 D1004  ; AX2 SERVO POSITION
      DMOV    D1250Z7 D1006  ; AX2 SERVO SPEED
47    LD      B131Z6
      DMOV    D1300Z7 D1008  ; AX3 SERVO POSITION
      DMOV    D1350Z7 D1010  ; AX3 SERVO SPEED
55    LD      B141Z6
      DMOV    D1400Z7 D1012  ; AX4 SERVO POSITION
      DMOV    D1450Z7 D1014  ; AX4 SERVO SPEED
63    LD      B151Z6
      DMOV    D1500Z7 D1016  ; AX5 SERVO POSITION
      DMOV    D1550Z7 D1018  ; AX5 SERVO SPEED
71    LD      B211Z6
      DMOV    D1600Z7 D1020  ; AX6 SERVO POSITION
      DMOV    D1650Z7 D1022  ; AX6 SERVO SPEED
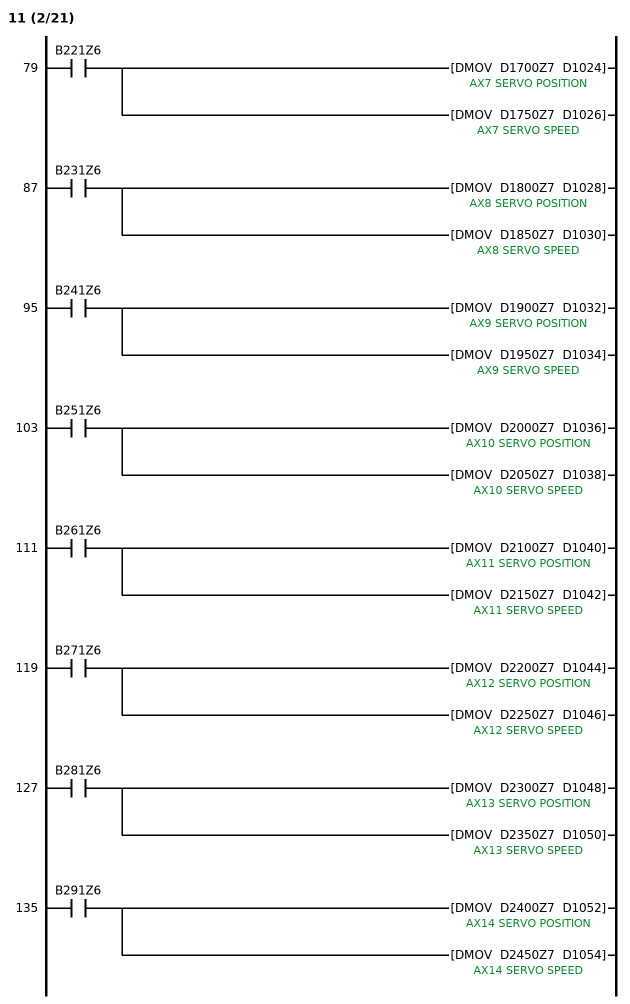
79    LD      B221Z6
      DMOV    D1700Z7 D1024  ; AX7 SERVO POSITION
      DMOV    D1750Z7 D1026  ; AX7 SERVO SPEED
87    LD      B231Z6
      DMOV    D1800Z7 D1028  ; AX8 SERVO POSITION
      DMOV    D1850Z7 D1030  ; AX8 SERVO SPEED
95    LD      B241Z6
      DMOV    D1900Z7 D1032  ; AX9 SERVO POSITION
      DMOV    D1950Z7 D1034  ; AX9 SERVO SPEED
103   LD      B251Z6
      DMOV    D2000Z7 D1036  ; AX10 SERVO POSITION
      DMOV    D2050Z7 D1038  ; AX10 SERVO SPEED
111   LD      B261Z6
      DMOV    D2100Z7 D1040  ; AX11 SERVO POSITION
      DMOV    D2150Z7 D1042  ; AX11 SERVO SPEED
119   LD      B271Z6
      DMOV    D2200Z7 D1044  ; AX12 SERVO POSITION
      DMOV    D2250Z7 D1046  ; AX12 SERVO SPEED
127   LD      B281Z6
      DMOV    D2300Z7 D1048  ; AX13 SERVO POSITION
      DMOV    D2350Z7 D1050  ; AX13 SERVO SPEED
135   LD      B291Z6
      DMOV    D2400Z7 D1052  ; AX14 SERVO POSITION
      DMOV    D2450Z7 D1054  ; AX14 SERVO SPEED
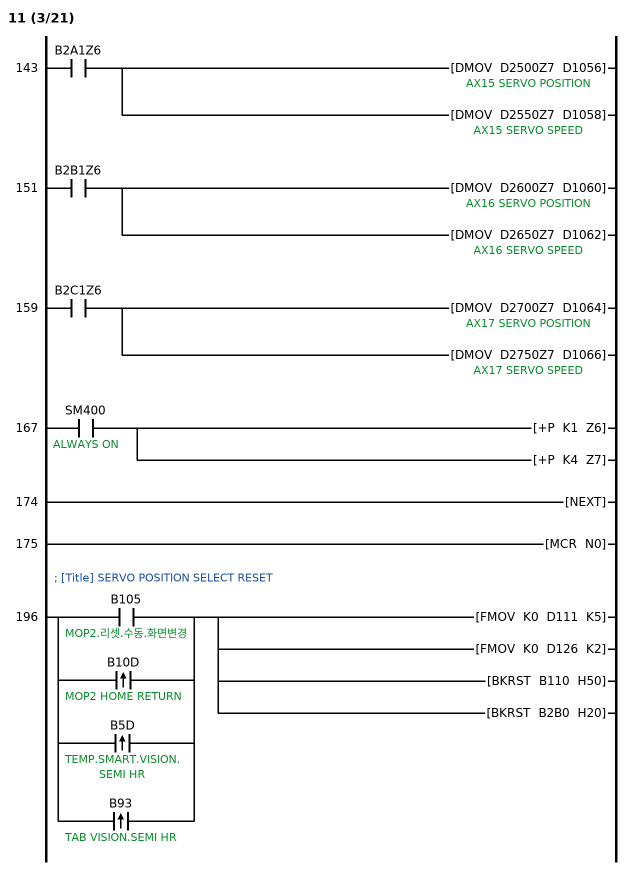
143   LD      B2A1Z6
      DMOV    D2500Z7 D1056  ; AX15 SERVO POSITION
      DMOV    D2550Z7 D1058  ; AX15 SERVO SPEED
151   LD      B2B1Z6
      DMOV    D2600Z7 D1060  ; AX16 SERVO POSITION
      DMOV    D2650Z7 D1062  ; AX16 SERVO SPEED
159   LD      B2C1Z6
      DMOV    D2700Z7 D1064  ; AX17 SERVO POSITION
      DMOV    D2750Z7 D1066  ; AX17 SERVO SPEED
167   LD      SM400  ; ALWAYS ON
      +P      K1 Z6
      +P      K4 Z7
174   NEXT
175   MCR     N0
; [Title] SERVO POSITION SELECT RESET
196   LD      B105  ; MOP2.리셋.수동.화면변경
      ORP     B10D  ; MOP2 HOME RETURN
      ORP     B5D  ; TEMP.SMART.VISION.SEMI HR
      ORP     B93  ; TAB VISION.SEMI HR
      FMOV    K0 D111 K5
      FMOV    K0 D126 K2
      BKRST   B110 H50
      BKRST   B2B0 H20
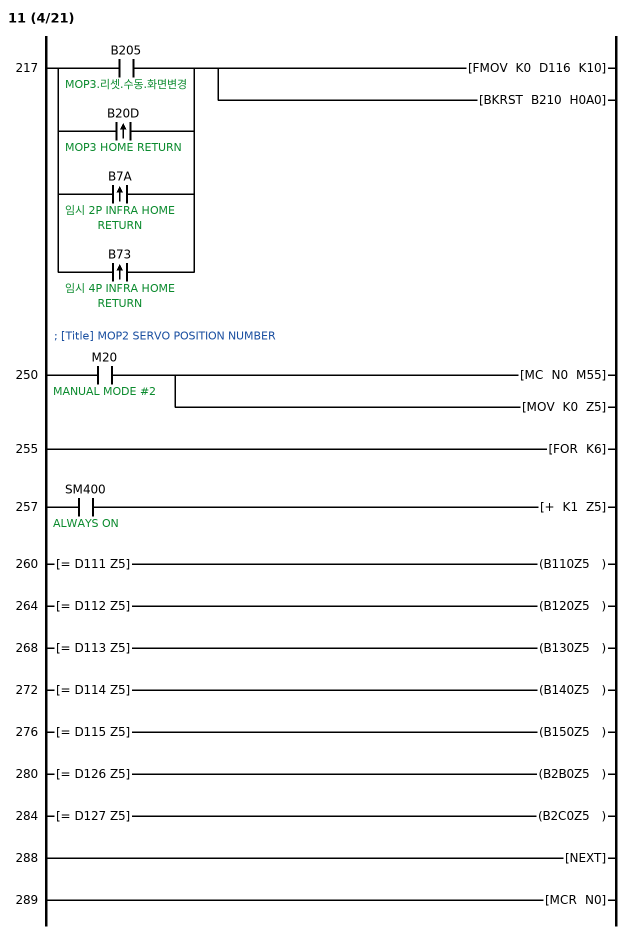
217   LD      B205  ; MOP3.리셋.수동.화면변경
      ORP     B20D  ; MOP3 HOME RETURN
      ORP     B7A  ; 임시 2P INFRA HOME RETURN
      ORP     B73  ; 임시 4P INFRA HOME RETURN
      FMOV    K0 D116 K10
      BKRST   B210 H0A0
; [Title] MOP2 SERVO POSITION NUMBER
250   LD      M20  ; MANUAL MODE #2
      MC      N0 M55
      MOV     K0 Z5
255   FOR     K6
257   LD      SM400  ; ALWAYS ON
      +       K1 Z5
260   LD=     D111 Z5
      OUT     B110Z5
264   LD=     D112 Z5
      OUT     B120Z5
268   LD=     D113 Z5
      OUT     B130Z5
272   LD=     D114 Z5
      OUT     B140Z5
276   LD=     D115 Z5
      OUT     B150Z5
280   LD=     D126 Z5
      OUT     B2B0Z5
284   LD=     D127 Z5
      OUT     B2C0Z5
288   NEXT
289   MCR     N0
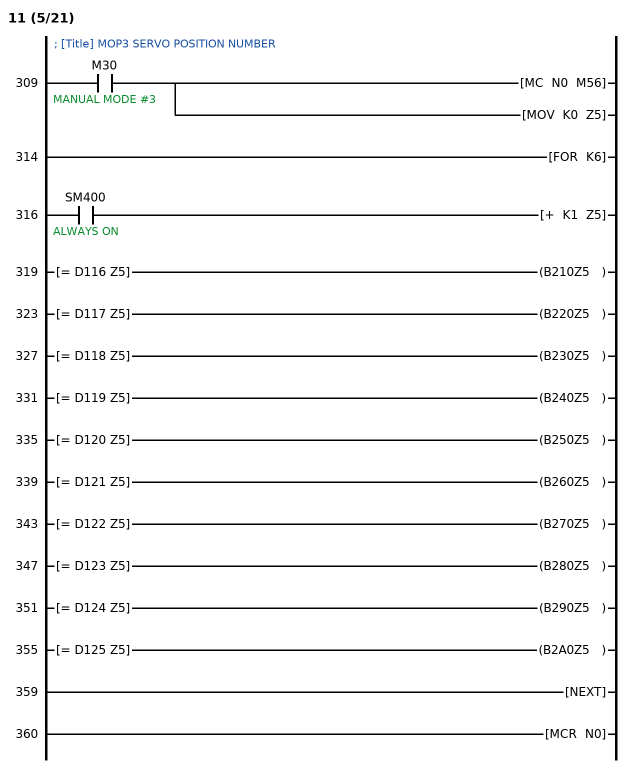
; [Title] MOP3 SERVO POSITION NUMBER
309   LD      M30  ; MANUAL MODE #3
      MC      N0 M56
      MOV     K0 Z5
314   FOR     K6
316   LD      SM400  ; ALWAYS ON
      +       K1 Z5
319   LD=     D116 Z5
      OUT     B210Z5
323   LD=     D117 Z5
      OUT     B220Z5
327   LD=     D118 Z5
      OUT     B230Z5
331   LD=     D119 Z5
      OUT     B240Z5
335   LD=     D120 Z5
      OUT     B250Z5
339   LD=     D121 Z5
      OUT     B260Z5
343   LD=     D122 Z5
      OUT     B270Z5
347   LD=     D123 Z5
      OUT     B280Z5
351   LD=     D124 Z5
      OUT     B290Z5
355   LD=     D125 Z5
      OUT     B2A0Z5
359   NEXT
360   MCR     N0
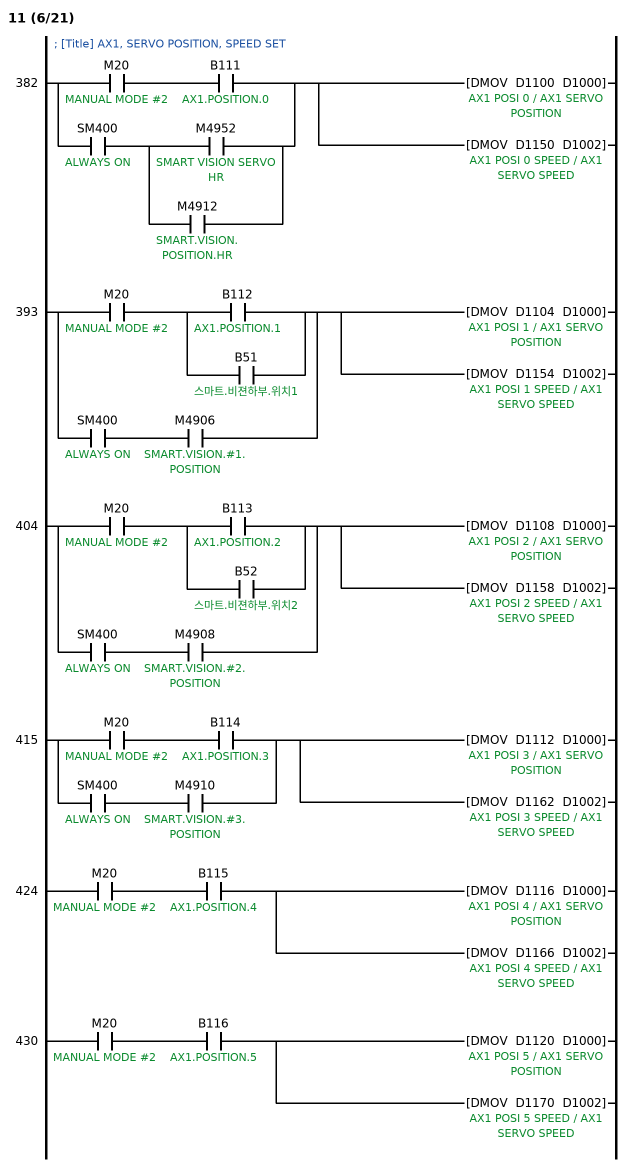
; [Title] AX1, SERVO POSITION, SPEED SET
382   LD      M20  ; MANUAL MODE #2
      AND     B111  ; AX1.POSITION.0
      LD      SM400  ; ALWAYS ON
      LD      M4952  ; SMART VISION SERVO HR
      OR      M4912  ; SMART.VISION.POSITION.HR
      ANB
      ORB
      DMOV    D1100 D1000  ; AX1 POSI 0
      DMOV    D1150 D1002  ; AX1 POSI 0 SPEED
393   LD      M20  ; MANUAL MODE #2
      LD      B112  ; AX1.POSITION.1
      OR      B51  ; 스마트.비젼하부.위치1
      ANB
      LD      SM400  ; ALWAYS ON
      AND     M4906  ; SMART.VISION.#1.POSITION
      ORB
      DMOV    D1104 D1000  ; AX1 POSI 1
      DMOV    D1154 D1002  ; AX1 POSI 1 SPEED
404   LD      M20  ; MANUAL MODE #2
      LD      B113  ; AX1.POSITION.2
      OR      B52  ; 스마트.비젼하부.위치2
      ANB
      LD      SM400  ; ALWAYS ON
      AND     M4908  ; SMART.VISION.#2.POSITION
      ORB
      DMOV    D1108 D1000  ; AX1 POSI 2
      DMOV    D1158 D1002  ; AX1 POSI 2 SPEED
415   LD      M20  ; MANUAL MODE #2
      AND     B114  ; AX1.POSITION.3
      LD      SM400  ; ALWAYS ON
      AND     M4910  ; SMART.VISION.#3.POSITION
      ORB
      DMOV    D1112 D1000  ; AX1 POSI 3
      DMOV    D1162 D1002  ; AX1 POSI 3 SPEED
424   LD      M20  ; MANUAL MODE #2
      AND     B115  ; AX1.POSITION.4
      DMOV    D1116 D1000  ; AX1 POSI 4
      DMOV    D1166 D1002  ; AX1 POSI 4 SPEED
430   LD      M20  ; MANUAL MODE #2
      AND     B116  ; AX1.POSITION.5
      DMOV    D1120 D1000  ; AX1 POSI 5
      DMOV    D1170 D1002  ; AX1 POSI 5 SPEED
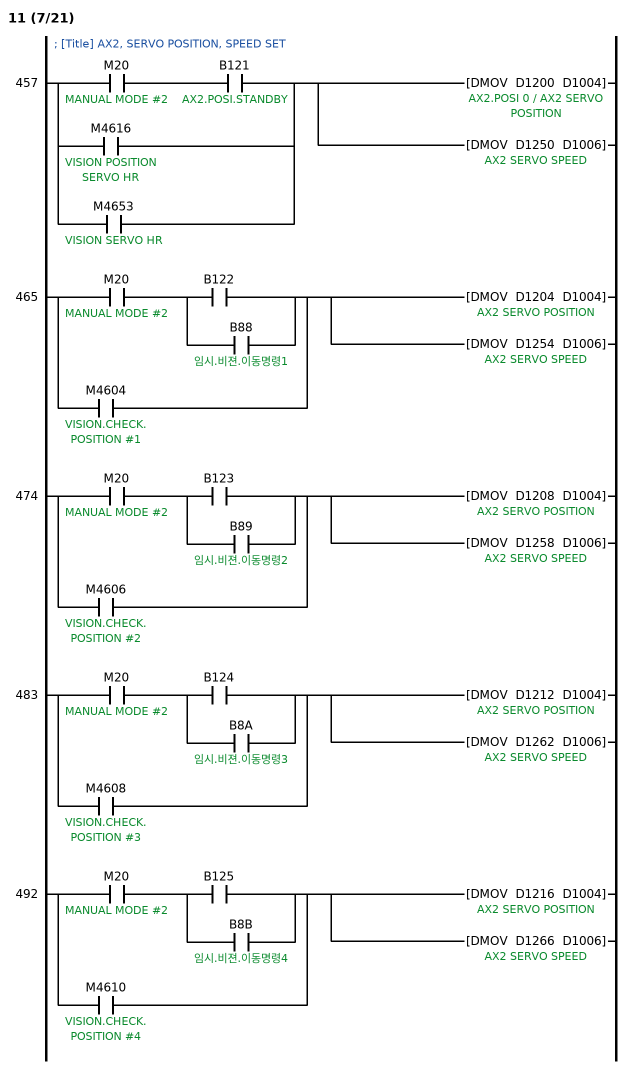
; [Title] AX2, SERVO POSITION, SPEED SET
457   LD      M20  ; MANUAL MODE #2
      AND     B121  ; AX2.POSI.STANDBY
      OR      M4616  ; VISION POSITION SERVO HR
      OR      M4653  ; VISION SERVO HR
      DMOV    D1200 D1004  ; AX2.POSI 0
      DMOV    D1250 D1006
465   LD      M20  ; MANUAL MODE #2
      LD      B122
      OR      B88  ; 임시.비젼.이동명령1
      ANB
      OR      M4604  ; VISION.CHECK.POSITION #1
      DMOV    D1204 D1004
      DMOV    D1254 D1006
474   LD      M20  ; MANUAL MODE #2
      LD      B123
      OR      B89  ; 임시.비젼.이동명령2
      ANB
      OR      M4606  ; VISION.CHECK.POSITION #2
      DMOV    D1208 D1004
      DMOV    D1258 D1006
483   LD      M20  ; MANUAL MODE #2
      LD      B124
      OR      B8A  ; 임시.비젼.이동명령3
      ANB
      OR      M4608  ; VISION.CHECK.POSITION #3
      DMOV    D1212 D1004
      DMOV    D1262 D1006
492   LD      M20  ; MANUAL MODE #2
      LD      B125
      OR      B8B  ; 임시.비젼.이동명령4
      ANB
      OR      M4610  ; VISION.CHECK.POSITION #4
      DMOV    D1216 D1004
      DMOV    D1266 D1006
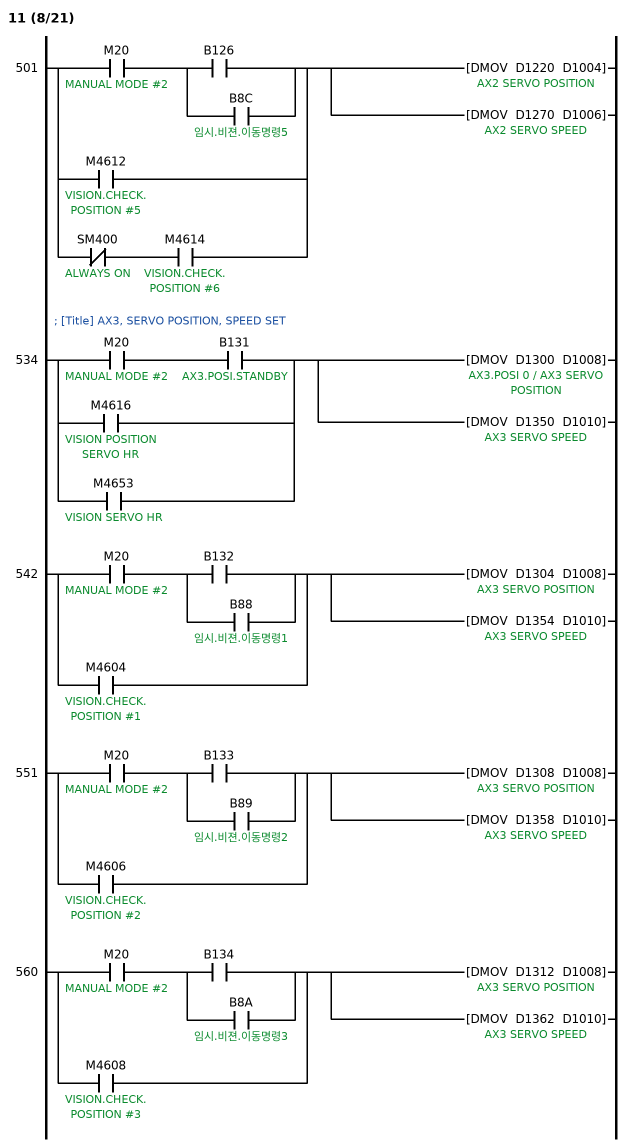
501   LD      M20  ; MANUAL MODE #2
      LD      B126
      OR      B8C  ; 임시.비젼.이동명령5
      ANB
      OR      M4612  ; VISION.CHECK.POSITION #5
      LDI     SM400  ; ALWAYS ON
      AND     M4614  ; VISION.CHECK.POSITION #6
      ORB
      DMOV    D1220 D1004
      DMOV    D1270 D1006
; [Title] AX3, SERVO POSITION, SPEED SET
534   LD      M20  ; MANUAL MODE #2
      AND     B131  ; AX3.POSI.STANDBY
      OR      M4616  ; VISION POSITION SERVO HR
      OR      M4653  ; VISION SERVO HR
      DMOV    D1300 D1008  ; AX3.POSI 0
      DMOV    D1350 D1010
542   LD      M20  ; MANUAL MODE #2
      LD      B132
      OR      B88  ; 임시.비젼.이동명령1
      ANB
      OR      M4604  ; VISION.CHECK.POSITION #1
      DMOV    D1304 D1008
      DMOV    D1354 D1010
551   LD      M20  ; MANUAL MODE #2
      LD      B133
      OR      B89  ; 임시.비젼.이동명령2
      ANB
      OR      M4606  ; VISION.CHECK.POSITION #2
      DMOV    D1308 D1008
      DMOV    D1358 D1010
560   LD      M20  ; MANUAL MODE #2
      LD      B134
      OR      B8A  ; 임시.비젼.이동명령3
      ANB
      OR      M4608  ; VISION.CHECK.POSITION #3
      DMOV    D1312 D1008
      DMOV    D1362 D1010
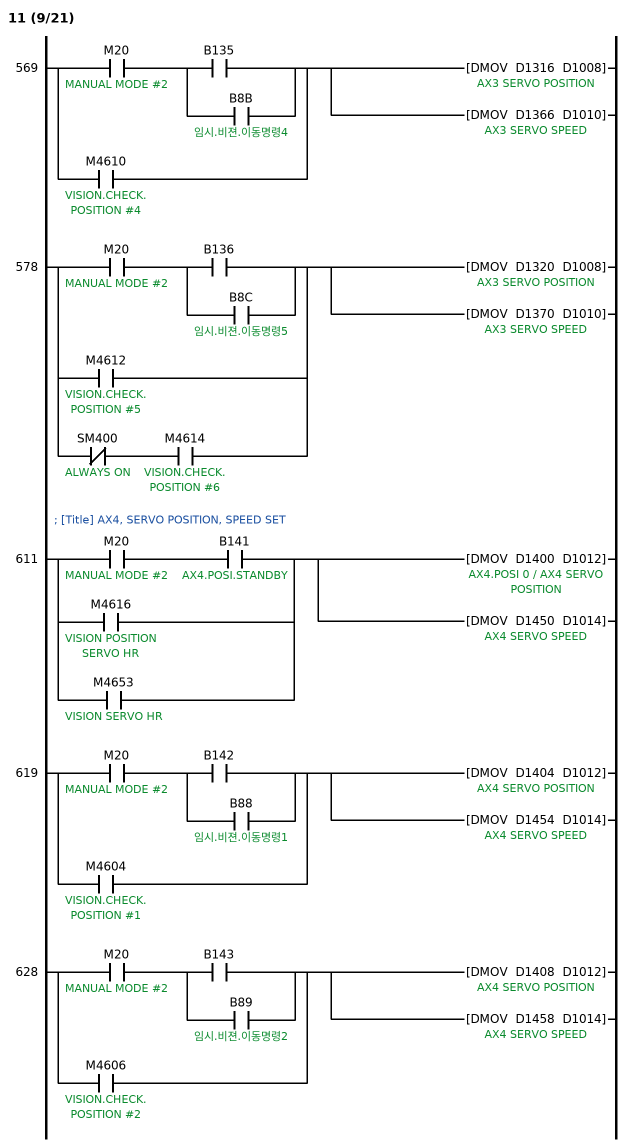
569   LD      M20  ; MANUAL MODE #2
      LD      B135
      OR      B8B  ; 임시.비젼.이동명령4
      ANB
      OR      M4610  ; VISION.CHECK.POSITION #4
      DMOV    D1316 D1008
      DMOV    D1366 D1010
578   LD      M20  ; MANUAL MODE #2
      LD      B136
      OR      B8C  ; 임시.비젼.이동명령5
      ANB
      OR      M4612  ; VISION.CHECK.POSITION #5
      LDI     SM400  ; ALWAYS ON
      AND     M4614  ; VISION.CHECK.POSITION #6
      ORB
      DMOV    D1320 D1008
      DMOV    D1370 D1010
; [Title] AX4, SERVO POSITION, SPEED SET
611   LD      M20  ; MANUAL MODE #2
      AND     B141  ; AX4.POSI.STANDBY
      OR      M4616  ; VISION POSITION SERVO HR
      OR      M4653  ; VISION SERVO HR
      DMOV    D1400 D1012  ; AX4.POSI 0
      DMOV    D1450 D1014
619   LD      M20  ; MANUAL MODE #2
      LD      B142
      OR      B88  ; 임시.비젼.이동명령1
      ANB
      OR      M4604  ; VISION.CHECK.POSITION #1
      DMOV    D1404 D1012
      DMOV    D1454 D1014
628   LD      M20  ; MANUAL MODE #2
      LD      B143
      OR      B89  ; 임시.비젼.이동명령2
      ANB
      OR      M4606  ; VISION.CHECK.POSITION #2
      DMOV    D1408 D1012
      DMOV    D1458 D1014
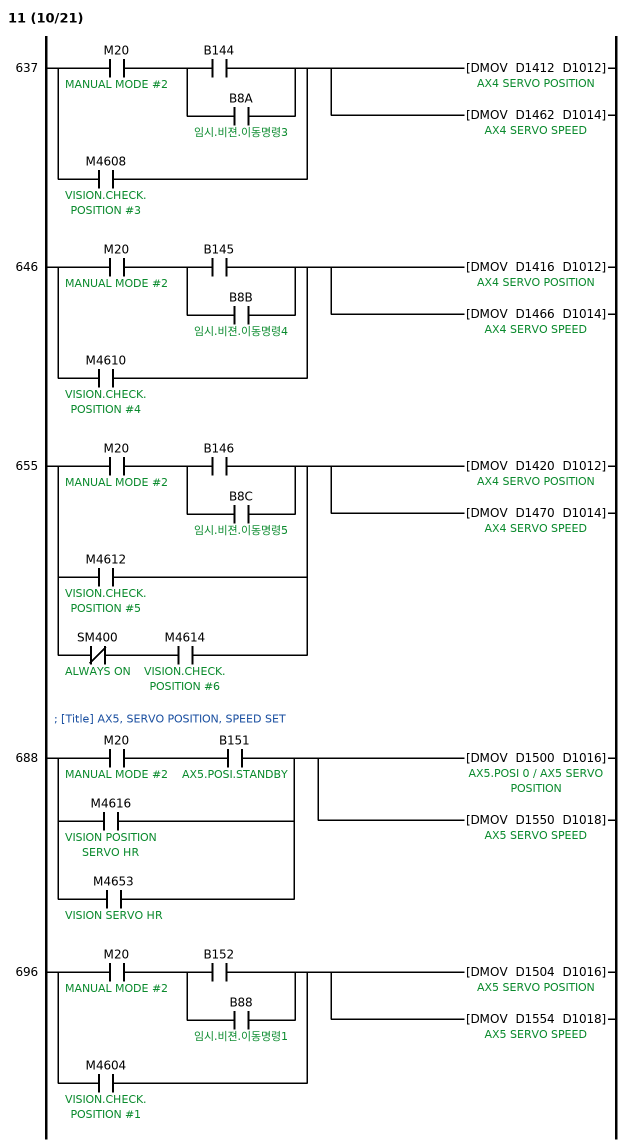
637   LD      M20  ; MANUAL MODE #2
      LD      B144
      OR      B8A  ; 임시.비젼.이동명령3
      ANB
      OR      M4608  ; VISION.CHECK.POSITION #3
      DMOV    D1412 D1012
      DMOV    D1462 D1014
646   LD      M20  ; MANUAL MODE #2
      LD      B145
      OR      B8B  ; 임시.비젼.이동명령4
      ANB
      OR      M4610  ; VISION.CHECK.POSITION #4
      DMOV    D1416 D1012
      DMOV    D1466 D1014
655   LD      M20  ; MANUAL MODE #2
      LD      B146
      OR      B8C  ; 임시.비젼.이동명령5
      ANB
      OR      M4612  ; VISION.CHECK.POSITION #5
      LDI     SM400  ; ALWAYS ON
      AND     M4614  ; VISION.CHECK.POSITION #6
      ORB
      DMOV    D1420 D1012
      DMOV    D1470 D1014
; [Title] AX5, SERVO POSITION, SPEED SET
688   LD      M20  ; MANUAL MODE #2
      AND     B151  ; AX5.POSI.STANDBY
      OR      M4616  ; VISION POSITION SERVO HR
      OR      M4653  ; VISION SERVO HR
      DMOV    D1500 D1016  ; AX5.POSI 0
      DMOV    D1550 D1018
696   LD      M20  ; MANUAL MODE #2
      LD      B152
      OR      B88  ; 임시.비젼.이동명령1
      ANB
      OR      M4604  ; VISION.CHECK.POSITION #1
      DMOV    D1504 D1016
      DMOV    D1554 D1018
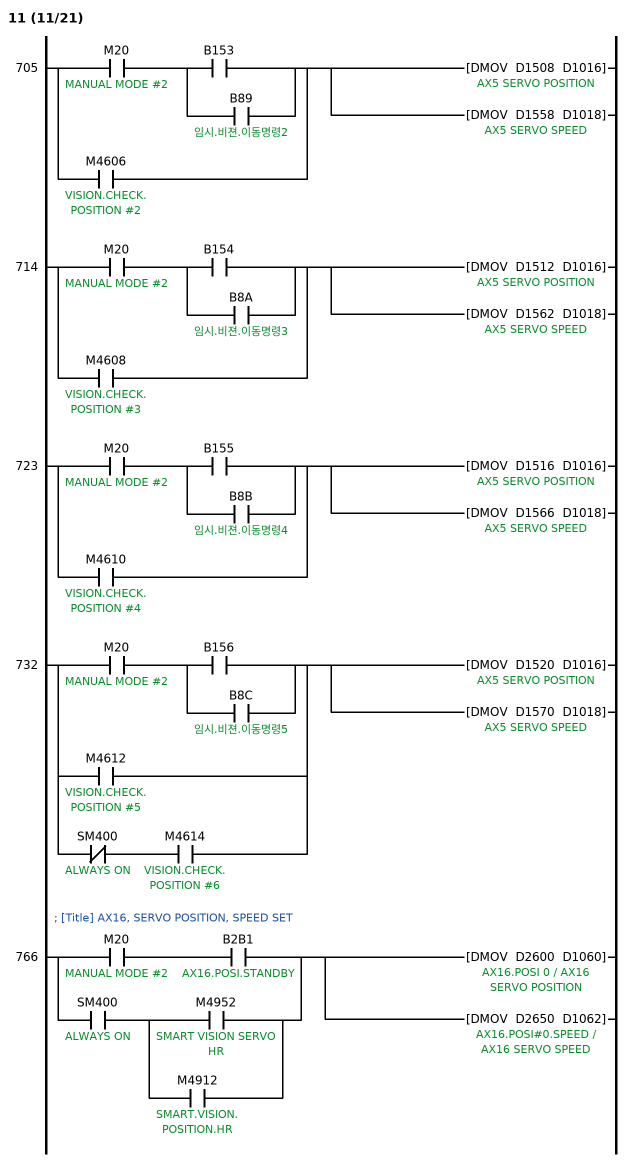
705   LD      M20  ; MANUAL MODE #2
      LD      B153
      OR      B89  ; 임시.비젼.이동명령2
      ANB
      OR      M4606  ; VISION.CHECK.POSITION #2
      DMOV    D1508 D1016
      DMOV    D1558 D1018
714   LD      M20  ; MANUAL MODE #2
      LD      B154
      OR      B8A  ; 임시.비젼.이동명령3
      ANB
      OR      M4608  ; VISION.CHECK.POSITION #3
      DMOV    D1512 D1016
      DMOV    D1562 D1018
723   LD      M20  ; MANUAL MODE #2
      LD      B155
      OR      B8B  ; 임시.비젼.이동명령4
      ANB
      OR      M4610  ; VISION.CHECK.POSITION #4
      DMOV    D1516 D1016
      DMOV    D1566 D1018
732   LD      M20  ; MANUAL MODE #2
      LD      B156
      OR      B8C  ; 임시.비젼.이동명령5
      ANB
      OR      M4612  ; VISION.CHECK.POSITION #5
      LDI     SM400  ; ALWAYS ON
      AND     M4614  ; VISION.CHECK.POSITION #6
      ORB
      DMOV    D1520 D1016
      DMOV    D1570 D1018
; [Title] AX16, SERVO POSITION, SPEED SET
766   LD      M20  ; MANUAL MODE #2
      AND     B2B1  ; AX16.POSI.STANDBY
      LD      SM400  ; ALWAYS ON
      LD      M4952  ; SMART VISION SERVO HR
      OR      M4912  ; SMART.VISION.POSITION.HR
      ANB
      ORB
      DMOV    D2600 D1060  ; AX16.POSI 0
      DMOV    D2650 D1062  ; AX16.POSI#0.SPEED
